C05348=1013.518,283.587,-142.989,169.129,53.074,160.196
C05349=1013.525,283.835,-143.018,169.134,53.067,160.195
C05350=1013.530,284.083,-143.047,169.141,53.060,160.195
C05351=1013.535,284.331,-143.077,169.146,53.053,160.195
C05352=1013.541,284.579,-143.107,169.151,53.046,160.194
C05353=1013.546,284.827,-143.137,169.157,53.039,160.194
C05354=1013.552,285.076,-143.167,169.163,53.032,160.193
C05355=1013.558,285.324,-143.197,169.169,53.025,160.193
C05356=1013.563,285.572,-143.227,169.174,53.018,160.192
C05357=1013.569,285.820,-143.257,169.181,53.011,160.192
C05358=1013.575,286.068,-143.287,169.186,53.004,160.192
C05359=1013.580,286.317,-143.316,169.192,52.997,160.191
C05360=1013.585,286.564,-143.346,169.198,52.990,160.191
C05361=1013.591,286.812,-143.376,169.204,52.983,160.191
C05362=1013.597,287.060,-143.406,169.209,52.976,160.190
C05363=1013.602,287.309,-143.436,169.216,52.969,160.190
C05364=1013.608,287.557,-143.466,169.222,52.962,160.190
C05365=1013.613,287.805,-143.496,169.227,52.955,160.189
C05366=1013.619,288.053,-143.526,169.233,52.949,160.189
C05367=1013.625,288.301,-143.556,169.239,52.941,160.188
C05368=1013.631,288.549,-143.586,169.245,52.935,160.188
C05369=1013.636,288.797,-143.617,169.250,52.928,160.187
C05370=1013.642,289.045,-143.646,169.257,52.921,160.187
C05371=1013.648,289.293,-143.676,169.263,52.915,160.187
C05372=1013.653,289.542,-143.706,169.268,52.908,160.187
C05373=1013.659,289.789,-143.736,169.274,52.901,160.186
C05374=1013.665,290.037,-143.767,169.280,52.894,160.186
C05375=1013.671,290.286,-143.798,169.286,52.887,160.186
C05376=1013.677,290.534,-143.827,169.292,52.881,160.185
C05377=1013.683,290.782,-143.858,169.298,52.873,160.185
C05378=1013.688,291.030,-143.888,169.304,52.867,160.185
C05379=1013.694,291.278,-143.918,169.310,52.861,160.184
C05380=1013.699,291.526,-143.949,169.316,52.854,160.184
C05381=1013.705,291.774,-143.979,169.322,52.847,160.184
C05382=1013.711,292.022,-144.009,169.328,52.840,160.183
C05383=1013.716,292.270,-144.040,169.334,52.834,160.183
C05384=1013.722,292.518,-144.070,169.339,52.827,160.183
C05385=1013.729,292.783,-144.103,169.346,52.820,160.182
C05386=1013.735,293.049,-144.136,169.353,52.813,160.182
C05387=1013.740,293.314,-144.169,169.359,52.806,160.182
C05388=1013.746,293.580,-144.202,169.365,52.799,160.181
C05389=1013.752,293.828,-144.233,169.372,52.792,160.181
C05390=1013.757,294.076,-144.264,169.377,52.786,160.181
C05391=1013.763,294.324,-144.295,169.383,52.780,160.181
C05392=1013.768,294.572,-144.326,169.389,52.773,160.180
C05393=1013.774,294.820,-144.356,169.395,52.767,160.180
C05394=1013.779,295.068,-144.387,169.402,52.760,160.180
C05395=1013.785,295.316,-144.418,169.407,52.754,160.179
C05396=1013.791,295.564,-144.450,169.413,52.747,160.179
C05397=1013.797,295.812,-144.480,169.419,52.741,160.179
C05398=1013.802,296.060,-144.511,169.425,52.734,160.179
C05399=1013.808,296.308,-144.542,169.431,52.728,160.178
C05400=1013.814,296.556,-144.573,169.438,52.721,160.178
C05401=1013.820,296.804,-144.604,169.444,52.716,160.178
C05402=1013.825,297.052,-144.635,169.450,52.709,160.178
C05403=1013.831,297.300,-144.666,169.455,52.703,160.177
C05404=1013.837,297.548,-144.698,169.461,52.696,160.177
C05405=1013.843,297.796,-144.728,169.468,52.690,160.177
C05406=1013.848,298.044,-144.759,169.474,52.683,160.177
C05407=1013.854,298.292,-144.790,169.480,52.678,160.177
C05408=1013.859,298.540,-144.821,169.486,52.671,160.176
C05409=1013.866,298.788,-144.853,169.492,52.665,160.176
C05410=1013.871,299.036,-144.884,169.499,52.658,160.176
C05411=1013.877,299.283,-144.915,169.505,52.652,160.176
C05412=1013.883,299.532,-144.946,169.511,52.646,160.175
C05413=1013.889,299.779,-144.977,169.517,52.640,160.175
C05414=1013.895,300.028,-145.008,169.523,52.634,160.175
C05415=1013.900,300.275,-145.040,169.529,52.627,160.175
C05416=1013.907,300.523,-145.072,169.535,52.621,160.175
C05417=1013.912,300.771,-145.102,169.542,52.615,160.174
C05418=1013.918,301.019,-145.134,169.548,52.609,160.174
C05419=1013.924,301.267,-145.165,169.553,52.602,160.174
C05420=1013.930,301.515,-145.196,169.560,52.597,160.174
C05421=1013.936,301.763,-145.228,169.566,52.590,160.174
C05422=1013.942,302.011,-145.258,169.573,52.584,160.174
C05423=1013.948,302.259,-145.290,169.579,52.578,160.173
C05424=1013.955,302.507,-145.322,169.585,52.572,160.173
C05425=1013.960,302.754,-145.353,169.591,52.566,160.173
C05426=1013.966,303.003,-145.384,169.597,52.559,160.173
C05427=1013.972,303.250,-145.416,169.604,52.553,160.173
C05428=1013.978,303.498,-145.447,169.610,52.547,160.172
C05429=1013.984,303.746,-145.479,169.616,52.541,160.172
C05430=1013.990,303.994,-145.510,169.622,52.535,160.172
C05431=1013.996,304.243,-145.542,169.629,52.529,160.172
C05432=1014.002,304.490,-145.573,169.635,52.523,160.172
C05433=1014.008,304.738,-145.605,169.641,52.517,160.171
C05434=1014.014,304.985,-145.636,169.647,52.511,160.171
C05435=1014.020,305.233,-145.668,169.653,52.505,160.171
C05436=1014.026,305.482,-145.700,169.660,52.498,160.171
C05437=1014.033,305.729,-145.731,169.667,52.493,160.171
C05438=1014.039,305.977,-145.763,169.672,52.486,160.171
C05439=1014.045,306.225,-145.794,169.679,52.481,160.171
C05440=1014.051,306.473,-145.826,169.686,52.475,160.171
C05441=1014.057,306.720,-145.857,169.692,52.468,160.170
C05442=1014.063,306.969,-145.889,169.698,52.463,160.170
C05443=1014.070,307.216,-145.921,169.704,52.457,160.170
C05444=1014.075,307.464,-145.953,169.711,52.451,160.170
C05445=1014.083,307.748,-145.989,169.719,52.444,160.170
C05446=1014.090,308.032,-146.025,169.725,52.437,160.170
C05447=1014.097,308.316,-146.062,169.733,52.430,160.170
C05448=1014.104,308.600,-146.098,169.740,52.424,160.169
C05449=1014.111,308.846,-146.130,169.746,52.418,160.169
C05450=1014.117,309.094,-146.161,169.753,52.412,160.169
C05451=1014.123,309.343,-146.193,169.760,52.406,160.169
C05452=1014.128,309.590,-146.226,169.766,52.401,160.169
C05453=1014.134,309.838,-146.258,169.772,52.395,160.169
C05454=1014.141,310.086,-146.291,169.779,52.389,160.169
C05455=1014.147,310.333,-146.324,169.785,52.384,160.169
C05456=1014.153,310.581,-146.356,169.792,52.379,160.169
C05457=1014.158,310.829,-146.389,169.798,52.373,160.169
C05458=1014.164,311.077,-146.421,169.804,52.367,160.169
C05459=1014.170,311.324,-146.453,169.811,52.362,160.169
C05460=1014.176,311.572,-146.486,169.817,52.356,160.169
C05461=1014.182,311.820,-146.518,169.824,52.350,160.169
C05462=1014.189,312.068,-146.551,169.831,52.345,160.169
C05463=1014.194,312.315,-146.584,169.837,52.339,160.169
C05464=1014.200,312.563,-146.616,169.843,52.333,160.169
C05465=1014.206,312.811,-146.649,169.850,52.328,160.169
C05466=1014.212,313.058,-146.681,169.856,52.323,160.169
C05467=1014.218,313.306,-146.714,169.863,52.317,160.169
C05468=1014.224,313.554,-146.746,169.869,52.311,160.169
C05469=1014.230,313.802,-146.780,169.876,52.306,160.169
C05470=1014.236,314.050,-146.812,169.883,52.300,160.169
C05471=1014.243,314.297,-146.845,169.889,52.295,160.169
C05472=1014.249,314.545,-146.878,169.896,52.290,160.169
C05473=1014.255,314.792,-146.911,169.902,52.284,160.169
C05474=1014.261,315.040,-146.944,169.909,52.278,160.169
C05475=1014.267,315.289,-146.976,169.915,52.273,160.169
C05476=1014.273,315.536,-147.009,169.922,52.268,160.169
C05477=1014.279,315.784,-147.041,169.928,52.263,160.169
C05478=1014.286,316.031,-147.074,169.936,52.257,160.169
C05479=1014.292,316.279,-147.107,169.942,52.252,160.169
C05480=1014.297,316.527,-147.140,169.949,52.246,160.169
C05481=1014.304,316.775,-147.173,169.955,52.241,160.169
C05482=1014.311,317.023,-147.206,169.962,52.236,160.169
C05483=1014.317,317.270,-147.239,169.968,52.231,160.169
C05484=1014.323,317.518,-147.272,169.975,52.225,160.169
C05485=1014.329,317.766,-147.305,169.982,52.220,160.169
C05486=1014.335,318.013,-147.338,169.989,52.214,160.169
C05487=1014.342,318.260,-147.371,169.995,52.209,160.169
C05488=1014.348,318.509,-147.404,170.002,52.203,160.169
C05489=1014.355,318.756,-147.437,170.008,52.198,160.169
C05490=1014.360,319.004,-147.470,170.015,52.193,160.169
C05491=1014.367,319.252,-147.503,170.022,52.187,160.169
C05492=1014.374,319.499,-147.537,170.029,52.182,160.169
C05493=1014.380,319.747,-147.570,170.036,52.177,160.170
C05494=1014.386,319.995,-147.602,170.042,52.172,160.169
C05495=1014.392,320.243,-147.636,170.049,52.167,160.170
C05496=1014.399,320.490,-147.669,170.056,52.162,160.170
C05497=1014.405,320.738,-147.702,170.063,52.156,160.170
C05498=1014.412,320.985,-147.735,170.070,52.151,160.170
C05499=1014.419,321.233,-147.769,170.076,52.146,160.170
C05500=1014.425,321.481,-147.802,170.083,52.141,160.170
C05501=1014.431,321.729,-147.835,170.090,52.136,160.170
C05502=1014.438,321.976,-147.869,170.096,52.131,160.170
C05503=1014.444,322.224,-147.901,170.104,52.125,160.170
C05504=1014.452,322.472,-147.935,170.110,52.120,160.170
C05505=1014.458,322.761,-147.974,170.118,52.114,160.171
C05506=1014.466,323.050,-148.013,170.126,52.108,160.171
C05507=1014.474,323.339,-148.052,170.135,52.102,160.171
C05508=1014.481,323.628,-148.091,170.143,52.096,160.171
C05509=1014.488,323.876,-148.124,170.149,52.091,160.171
C05510=1014.495,324.123,-148.158,170.156,52.086,160.171
C05511=1014.501,324.372,-148.191,170.164,52.081,160.171
C05512=1014.507,324.619,-148.225,170.170,52.076,160.172
C05513=1014.515,324.867,-148.259,170.177,52.071,160.172
C05514=1014.521,325.114,-148.291,170.184,52.066,160.172
C05515=1014.528,325.362,-148.325,170.192,52.061,160.172
C05516=1014.535,325.609,-148.359,170.198,52.056,160.172
C05517=1014.541,325.857,-148.392,170.205,52.051,160.172
C05518=1014.547,326.104,-148.426,170.212,52.046,160.172
C05519=1014.554,326.352,-148.460,170.219,52.042,160.173
C05520=1014.560,326.600,-148.495,170.226,52.037,160.173
C05521=1014.567,326.847,-148.528,170.233,52.031,160.173
C05522=1014.573,327.095,-148.563,170.240,52.026,160.173
C05523=1014.579,327.343,-148.597,170.247,52.022,160.174
C05524=1014.586,327.590,-148.631,170.254,52.017,160.174
C05525=1014.593,327.838,-148.665,170.261,52.012,160.174
C05526=1014.599,328.085,-148.699,170.268,52.008,160.174
C05527=1014.606,328.333,-148.733,170.275,52.003,160.174
C05528=1014.612,328.580,-148.768,170.283,51.998,160.175
C05529=1014.619,328.828,-148.802,170.290,51.993,160.175
C05530=1014.626,329.075,-148.836,170.296,51.988,160.175
C05531=1014.632,329.323,-148.870,170.303,51.984,160.175
C05532=1014.638,329.571,-148.904,170.310,51.979,160.175
C05533=1014.645,329.818,-148.938,170.318,51.974,160.176
C05534=1014.652,330.066,-148.973,170.325,51.969,160.176
C05535=1014.658,330.313,-149.007,170.332,51.965,160.176
C05536=1014.665,330.561,-149.041,170.339,51.960,160.176
C05537=1014.672,330.809,-149.076,170.346,51.956,160.177
C05538=1014.678,331.056,-149.111,170.353,51.951,160.177
C05539=1014.686,331.304,-149.145,170.361,51.946,160.177
C05540=1014.691,331.551,-149.179,170.368,51.942,160.178
C05541=1014.698,331.798,-149.214,170.375,51.937,160.178
C05542=1014.705,332.046,-149.248,170.382,51.933,160.178
C05543=1014.712,332.293,-149.283,170.389,51.928,160.178
C05544=1014.719,332.541,-149.317,170.397,51.923,160.178
C05545=1014.725,332.789,-149.352,170.404,51.919,160.179
C05546=1014.731,333.036,-149.386,170.411,51.914,160.179
C05547=1014.738,333.283,-149.421,170.418,51.910,160.179
C05548=1014.745,333.531,-149.457,170.425,51.905,160.180
C05549=1014.751,333.779,-149.491,170.433,51.901,160.180
C05550=1014.759,334.026,-149.526,170.440,51.896,160.180
C05551=1014.766,334.273,-149.561,170.448,51.892,160.181
C05552=1014.772,334.521,-149.595,170.455,51.888,160.181
C05553=1014.779,334.769,-149.630,170.462,51.883,160.181
C05554=1014.786,335.016,-149.665,170.470,51.878,160.182
C05555=1014.792,335.263,-149.700,170.477,51.874,160.182
C05556=1014.799,335.511,-149.735,170.484,51.870,160.182
C05557=1014.806,335.759,-149.770,170.491,51.865,160.182
C05558=1014.812,336.006,-149.805,170.498,51.861,160.183
C05559=1014.819,336.253,-149.840,170.506,51.856,160.183
C05560=1014.826,336.501,-149.875,170.513,51.852,160.184
C05561=1014.833,336.748,-149.911,170.521,51.848,160.184
C05562=1014.839,336.995,-149.946,170.528,51.843,160.184
C05563=1014.846,337.243,-149.980,170.535,51.839,160.185
C05564=1014.853,337.491,-150.015,170.543,51.834,160.185
C05565=1014.861,337.776,-150.056,170.551,51.830,160.185
C05566=1014.869,338.060,-150.097,170.560,51.825,160.186
C05567=1014.877,338.345,-150.136,170.569,51.820,160.186
C05568=1014.885,338.630,-150.177,170.578,51.815,160.187
C05569=1014.892,338.878,-150.212,170.585,51.811,160.187
C05570=1014.899,339.125,-150.248,170.592,51.807,160.187
C05571=1014.905,339.372,-150.284,170.600,51.803,160.188
C05572=1014.912,339.619,-150.319,170.608,51.798,160.188
C05573=1014.919,339.867,-150.355,170.615,51.794,160.189
C05574=1014.926,340.114,-150.390,170.623,51.790,160.189
C05575=1014.933,340.362,-150.426,170.630,51.786,160.190
C05576=1014.940,340.609,-150.461,170.638,51.781,160.190
C05577=1014.946,340.856,-150.497,170.645,51.778,160.191
C05578=1014.954,341.104,-150.533,170.653,51.773,160.191
C05579=1014.960,341.351,-150.568,170.660,51.770,160.191
C05580=1014.967,341.598,-150.604,170.668,51.765,160.192
C05581=1014.975,341.846,-150.639,170.675,51.761,160.192
C05582=1014.981,342.093,-150.676,170.683,51.757,160.193
C05583=1014.988,342.341,-150.711,170.690,51.753,160.193
C05584=1014.996,342.588,-150.747,170.699,51.749,160.194
C05585=1015.002,342.835,-150.782,170.706,51.745,160.194
C05586=1015.009,343.083,-150.819,170.714,51.741,160.194
C05587=1015.016,343.330,-150.855,170.721,51.737,160.195
C05588=1015.023,343.577,-150.890,170.729,51.733,160.195
C05589=1015.030,343.825,-150.927,170.737,51.729,160.196
C05590=1015.037,344.072,-150.963,170.744,51.726,160.197
C05591=1015.044,344.319,-150.998,170.753,51.721,160.197
C05592=1015.052,344.567,-151.034,170.760,51.717,160.197
C05593=1015.058,344.814,-151.070,170.768,51.714,160.198
C05594=1015.066,345.061,-151.107,170.776,51.709,160.198
C05595=1015.072,345.309,-151.142,170.783,51.705,160.199
C05596=1015.080,345.556,-151.178,170.791,51.702,160.199
C05597=1015.086,345.803,-151.214,170.799,51.698,160.200
C05598=1015.094,346.050,-151.251,170.807,51.694,160.201
C05599=1015.101,346.297,-151.286,170.814,51.690,160.201
C05600=1015.108,346.545,-151.323,170.822,51.686,160.201
C05601=1015.116,346.792,-151.359,170.830,51.682,160.202
C05602=1015.122,347.039,-151.396,170.838,51.679,160.203
C05603=1015.130,347.287,-151.432,170.846,51.675,160.203
C05604=1015.137,347.534,-151.468,170.854,51.671,160.204
C05605=1015.144,347.781,-151.505,170.862,51.667,160.204
C05606=1015.151,348.028,-151.541,170.869,51.664,160.205
C05607=1015.158,348.276,-151.577,170.878,51.660,160.206
C05608=1015.165,348.523,-151.615,170.886,51.656,160.206
C05609=1015.172,348.770,-151.651,170.893,51.652,160.207
C05610=1015.179,349.018,-151.688,170.902,51.649,160.207
C05611=1015.187,349.265,-151.724,170.909,51.645,160.208
C05612=1015.193,349.511,-151.761,170.917,51.641,160.208
C05613=1015.201,349.759,-151.797,170.926,51.638,160.209
C05614=1015.208,350.007,-151.834,170.933,51.634,160.210
C05615=1015.216,350.253,-151.871,170.942,51.630,160.210
C05616=1015.222,350.500,-151.907,170.950,51.627,160.211
C05617=1015.230,350.747,-151.944,170.957,51.623,160.211
C05618=1015.237,350.995,-151.981,170.966,51.620,160.212
C05619=1015.245,351.243,-152.017,170.974,51.616,160.213
C05620=1015.252,351.490,-152.055,170.981,51.612,160.213
C05621=1015.259,351.736,-152.091,170.990,51.609,160.214
C05622=1015.266,351.984,-152.128,170.998,51.605,160.215
C05623=1015.274,352.231,-152.166,171.006,51.601,160.215
C05624=1015.281,352.478,-152.202,171.014,51.598,160.216
C05625=1015.290,352.760,-152.244,171.024,51.594,160.217
C05626=1015.299,353.042,-152.287,171.033,51.590,160.217
C05627=1015.307,353.325,-152.329,171.043,51.586,160.218
C05628=1015.315,353.607,-152.371,171.052,51.582,160.219
C05629=1015.322,353.854,-152.408,171.060,51.579,160.220
C05630=1015.330,354.100,-152.445,171.068,51.575,160.220
C05631=1015.337,354.348,-152.483,171.077,51.572,160.221
C05632=1015.344,354.595,-152.520,171.084,51.568,160.222
C05633=1015.352,354.842,-152.558,171.093,51.565,160.222
C05634=1015.360,355.089,-152.595,171.101,51.561,160.223
C05635=1015.367,355.336,-152.632,171.110,51.558,160.224
C05636=1015.374,355.584,-152.669,171.118,51.555,160.224
C05637=1015.382,355.831,-152.707,171.126,51.551,160.225
C05638=1015.390,356.078,-152.745,171.134,51.548,160.226
C05639=1015.397,356.325,-152.782,171.143,51.545,160.227
C05640=1015.405,356.572,-152.820,171.151,51.542,160.227
C05641=1015.412,356.819,-152.857,171.160,51.538,160.228
C05642=1015.420,357.066,-152.894,171.168,51.535,160.229
C05643=1015.427,357.313,-152.932,171.177,51.532,160.230
C05644=1015.434,357.560,-152.969,171.185,51.529,160.230
C05645=1015.442,357.807,-153.008,171.194,51.525,160.231
C05646=1015.450,358.054,-153.045,171.202,51.522,160.232
C05647=1015.458,358.301,-153.082,171.211,51.519,160.233
C05648=1015.465,358.548,-153.120,171.219,51.516,160.233
C05649=1015.472,358.795,-153.158,171.227,51.512,160.234
C05650=1015.480,359.043,-153.196,171.236,51.510,160.235
C05651=1015.488,359.289,-153.234,171.245,51.506,160.236
C05652=1015.495,359.536,-153.272,171.253,51.503,160.237
C05653=1015.503,359.783,-153.310,171.262,51.500,160.237
C05654=1015.510,360.030,-153.348,171.270,51.497,160.238
C05655=1015.518,360.277,-153.386,171.279,51.494,160.239
C05656=1015.525,360.524,-153.424,171.287,51.491,160.240
C05657=1015.533,360.771,-153.462,171.296,51.487,160.241
C05658=1015.541,361.018,-153.501,171.304,51.485,160.242
C05659=1015.548,361.265,-153.539,171.313,51.482,160.242
C05660=1015.556,361.512,-153.576,171.322,51.478,160.243
C05661=1015.563,361.759,-153.616,171.330,51.475,160.244
C05662=1015.571,362.006,-153.654,171.339,51.472,160.245
C05663=1015.579,362.253,-153.692,171.347,51.469,160.246
C05664=1015.586,362.500,-153.730,171.356,51.466,160.247
C05665=1015.594,362.747,-153.768,171.366,51.463,160.248
C05666=1015.602,362.994,-153.807,171.374,51.460,160.248
C05667=1015.609,363.240,-153.845,171.383,51.457,160.249
C05668=1015.617,363.488,-153.884,171.391,51.455,160.250
C05669=1015.625,363.734,-153.922,171.400,51.451,160.251
C05670=1015.633,363.981,-153.960,171.410,51.449,160.252
C05671=1015.641,364.228,-153.999,171.418,51.446,160.253
C05672=1015.649,364.475,-154.037,171.427,51.443,160.254
C05673=1015.657,364.722,-154.076,171.436,51.440,160.255
C05674=1015.665,364.969,-154.114,171.444,51.437,160.256
C05675=1015.673,365.216,-154.153,171.453,51.434,160.256
C05676=1015.680,365.463,-154.191,171.463,51.431,160.257
C05677=1015.689,365.709,-154.230,171.471,51.429,160.258
C05678=1015.696,365.957,-154.270,171.480,51.425,160.259
C05679=1015.704,366.203,-154.308,171.489,51.423,160.260
C05680=1015.712,366.450,-154.346,171.499,51.420,160.261
C05681=1015.720,366.697,-154.386,171.507,51.417,160.262
C05682=1015.728,366.944,-154.424,171.516,51.414,160.263
C05683=1015.736,367.191,-154.463,171.526,51.412,160.264
C05684=1015.744,367.437,-154.502,171.534,51.409,160.265
C05685=1015.753,367.727,-154.548,171.545,51.406,160.266
C05686=1015.763,368.017,-154.594,171.556,51.403,160.267
C05687=1015.772,368.307,-154.639,171.566,51.400,160.268
C05688=1015.781,368.596,-154.685,171.577,51.396,160.270
C05689=1015.789,368.843,-154.725,171.586,51.394,160.271
C05690=1015.797,369.090,-154.764,171.595,51.391,160.272
C05691=1015.806,369.336,-154.804,171.605,51.388,160.273
C05692=1015.813,369.584,-154.843,171.613,51.386,160.274
C05693=1015.821,369.831,-154.882,171.623,51.383,160.275
C05694=1015.829,370.077,-154.922,171.632,51.380,160.276
C05695=1015.837,370.323,-154.961,171.642,51.378,160.277
C05696=1015.845,370.570,-155.000,171.651,51.376,160.278
C05697=1015.853,370.817,-155.040,171.660,51.373,160.279
C05698=1015.861,371.064,-155.079,171.669,51.371,160.280
C05699=1015.869,371.311,-155.119,171.678,51.368,160.281
C05700=1015.878,371.558,-155.158,171.688,51.366,160.282
C05701=1015.886,371.804,-155.197,171.698,51.363,160.283
C05702=1015.894,372.051,-155.237,171.707,51.360,160.284
C05703=1015.902,372.298,-155.277,171.715,51.358,160.285
C05704=1015.911,372.544,-155.317,171.725,51.356,160.287
C05705=1015.919,372.791,-155.357,171.735,51.353,160.288
C05706=1015.927,373.037,-155.396,171.744,51.351,160.289
C05707=1015.935,373.284,-155.436,171.754,51.348,160.290
C05708=1015.943,373.531,-155.475,171.763,51.346,160.291
C05709=1015.952,373.778,-155.515,171.773,51.343,160.292
C05710=1015.960,374.024,-155.556,171.782,51.341,160.293
C05711=1015.969,374.271,-155.595,171.792,51.339,160.294
C05712=1015.977,374.518,-155.635,171.801,51.336,160.295
C05713=1015.985,374.764,-155.675,171.811,51.334,160.297
C05714=1015.994,375.011,-155.715,171.821,51.332,160.298
C05715=1016.002,375.258,-155.754,171.830,51.329,160.299
C05716=1016.011,375.504,-155.795,171.840,51.327,160.300
C05717=1016.019,375.751,-155.834,171.850,51.325,160.302
C05718=1016.027,375.998,-155.875,171.859,51.322,160.303
C05719=1016.036,376.244,-155.915,171.868,51.320,160.304
C05720=1016.044,376.491,-155.955,171.878,51.318,160.305
C05721=1016.052,376.737,-155.996,171.888,51.316,160.306
C05722=1016.060,376.984,-156.037,171.898,51.314,160.307
C05723=1016.069,377.230,-156.077,171.907,51.311,160.308
C05724=1016.077,377.476,-156.118,171.917,51.309,160.310
C05725=1016.085,377.724,-156.158,171.927,51.307,160.311
C05726=1016.093,377.970,-156.199,171.937,51.304,160.312
C05727=1016.102,378.216,-156.239,171.947,51.302,160.314
C05728=1016.111,378.463,-156.280,171.957,51.300,160.315
C05729=1016.119,378.709,-156.320,171.967,51.298,160.316
C05730=1016.128,378.956,-156.361,171.977,51.296,160.317
C05731=1016.136,379.202,-156.401,171.986,51.294,160.319
C05732=1016.145,379.449,-156.442,171.997,51.292,160.320
C05733=1016.153,379.696,-156.483,172.006,51.290,160.321
C05734=1016.163,379.942,-156.524,172.016,51.288,160.323
C05735=1016.171,380.188,-156.565,172.026,51.286,160.324
C05736=1016.179,380.435,-156.606,172.036,51.284,160.325
C05737=1016.187,380.681,-156.646,172.047,51.282,160.327
C05738=1016.197,380.928,-156.687,172.057,51.280,160.328
C05739=1016.206,381.174,-156.728,172.067,51.278,160.329
C05740=1016.214,381.421,-156.769,172.076,51.276,160.330
C05741=1016.222,381.668,-156.810,172.087,51.274,160.332
C05742=1016.231,381.913,-156.851,172.097,51.272,160.333
C05743=1016.240,382.160,-156.892,172.108,51.270,160.335
C05744=1016.249,382.407,-156.933,172.117,51.268,160.336
C05745=1016.260,382.719,-156.985,172.130,51.265,160.338
C05746=1016.271,383.031,-157.037,172.143,51.263,160.339
C05747=1016.282,383.343,-157.090,172.156,51.261,160.341
C05748=1016.294,383.656,-157.141,172.169,51.258,160.343
C05749=1016.303,383.903,-157.183,172.179,51.256,160.344
C05750=1016.311,384.148,-157.224,172.190,51.254,160.346
C05751=1016.321,384.395,-157.265,172.201,51.253,160.347
C05752=1016.330,384.641,-157.307,172.210,51.251,160.348
C05753=1016.338,384.888,-157.348,172.222,51.249,160.350
C05754=1016.347,385.134,-157.390,172.232,51.247,160.351
C05755=1016.356,385.381,-157.432,172.242,51.246,160.353
C05756=1016.365,385.627,-157.473,172.253,51.243,160.354
C05757=1016.374,385.873,-157.515,172.263,51.242,160.356
C05758=1016.383,386.120,-157.557,172.273,51.240,160.357
C05759=1016.392,386.366,-157.599,172.284,51.238,160.359
C05760=1016.401,386.612,-157.640,172.295,51.237,160.360
C05761=1016.409,386.858,-157.682,172.305,51.235,160.362
C05762=1016.419,387.105,-157.724,172.316,51.234,160.363
C05763=1016.428,387.351,-157.765,172.326,51.232,160.365
C05764=1016.437,387.598,-157.807,172.337,51.230,160.366
C05765=1016.446,387.844,-157.850,172.348,51.229,160.368
C05766=1016.455,388.090,-157.891,172.359,51.227,160.369
C05767=1016.464,388.336,-157.934,172.369,51.226,160.371
C05768=1016.473,388.582,-157.975,172.380,51.224,160.372
C05769=1016.482,388.828,-158.017,172.391,51.222,160.374
C05770=1016.490,389.074,-158.060,172.401,51.221,160.375
C05771=1016.499,389.321,-158.102,172.413,51.220,160.377
C05772=1016.509,389.567,-158.145,172.423,51.218,160.378
C05773=1016.519,389.813,-158.187,172.434,51.216,160.380
C05774=1016.527,390.059,-158.229,172.446,51.215,160.382
C05775=1016.537,390.305,-158.271,172.456,51.213,160.383
C05776=1016.547,390.552,-158.314,172.467,51.212,160.385
C05777=1016.555,390.798,-158.356,172.478,51.210,160.386
C05778=1016.564,391.044,-158.399,172.489,51.209,160.388
C05779=1016.574,391.290,-158.442,172.499,51.208,160.390
C05780=1016.583,391.536,-158.484,172.511,51.206,160.391
C05781=1016.592,391.783,-158.526,172.522,51.204,160.393
C05782=1016.602,392.029,-158.569,172.533,51.203,160.395
C05783=1016.610,392.275,-158.612,172.544,51.202,160.396
C05784=1016.620,392.522,-158.654,172.555,51.200,160.398
C05785=1016.630,392.767,-158.698,172.566,51.199,160.400
C05786=1016.639,393.012,-158.740,172.578,51.198,160.401
C05787=1016.648,393.259,-158.783,172.589,51.197,160.403
C05788=1016.657,393.505,-158.826,172.599,51.195,160.405
C05789=1016.667,393.751,-158.869,172.611,51.194,160.406
C05790=1016.676,393.997,-158.912,172.623,51.192,160.408
C05791=1016.686,394.243,-158.955,172.633,51.192,160.410
C05792=1016.696,394.490,-158.998,172.645,51.190,160.412
C05793=1016.704,394.736,-159.041,172.656,51.189,160.413
C05794=1016.714,394.982,-159.084,172.668,51.188,160.415
C05795=1016.724,395.227,-159.127,172.680,51.186,160.417
C05796=1016.733,395.473,-159.171,172.690,51.185,160.419
C05797=1016.743,395.720,-159.214,172.702,51.184,160.420
C05798=1016.752,395.965,-159.257,172.713,51.183,160.422
C05799=1016.761,396.212,-159.300,172.725,51.182,160.424
C05800=1016.772,396.458,-159.344,172.737,51.181,160.426
C05801=1016.782,396.703,-159.387,172.749,51.179,160.428
C05802=1016.790,396.949,-159.430,172.760,51.178,160.429
C05803=1016.800,397.195,-159.474,172.771,51.178,160.431
C05804=1016.810,397.441,-159.518,172.783,51.176,160.433
C05805=1016.824,397.787,-159.579,172.799,51.175,160.436
C05806=1016.837,398.133,-159.641,172.816,51.174,160.438
C05807=1016.851,398.479,-159.702,172.832,51.172,160.441
C05808=1016.865,398.826,-159.764,172.849,51.170,160.443
C05809=1016.874,399.071,-159.807,172.861,51.170,160.445
C05810=1016.884,399.318,-159.851,172.873,51.169,160.447
C05811=1016.894,399.563,-159.895,172.884,51.168,160.449
C05812=1016.904,399.809,-159.940,172.896,51.167,160.451
C05813=1016.914,400.055,-159.983,172.909,51.166,160.453
C05814=1016.923,400.301,-160.027,172.921,51.164,160.455
C05815=1016.934,400.547,-160.073,172.933,51.164,160.457
C05816=1016.943,400.793,-160.117,172.945,51.163,160.459
C05817=1016.953,401.038,-160.161,172.957,51.162,160.461
C05818=1016.963,401.285,-160.205,172.969,51.161,160.463
C05819=1016.973,401.530,-160.250,172.981,51.161,160.465
C05820=1016.983,401.776,-160.293,172.993,51.160,160.467
C05821=1016.992,402.021,-160.338,173.005,51.159,160.469
C05822=1017.002,402.268,-160.382,173.018,51.158,160.471
C05823=1017.012,402.514,-160.427,173.030,51.157,160.473
C05824=1017.023,402.759,-160.472,173.042,51.156,160.475
C05825=1017.032,403.004,-160.517,173.054,51.156,160.477
C05826=1017.042,403.251,-160.561,173.066,51.156,160.479
C05827=1017.053,403.497,-160.605,173.079,51.154,160.481
C05828=1017.062,403.742,-160.650,173.091,51.154,160.483
C05829=1017.072,403.988,-160.695,173.103,51.153,160.485
C05830=1017.083,404.233,-160.739,173.117,51.152,160.487
C05831=1017.093,404.479,-160.784,173.129,51.152,160.489
C05832=1017.103,404.724,-160.829,173.141,51.151,160.491
C05833=1017.113,404.971,-160.874,173.154,51.150,160.493
C05834=1017.123,405.216,-160.919,173.166,51.149,160.495
C05835=1017.134,405.461,-160.964,173.178,51.149,160.498
C05836=1017.144,405.707,-161.009,173.192,51.149,160.500
C05837=1017.155,405.953,-161.054,173.204,51.148,160.502
C05838=1017.165,406.198,-161.099,173.217,51.147,160.504
C05839=1017.175,406.444,-161.145,173.229,51.147,160.506
C05840=1017.186,406.690,-161.189,173.242,51.146,160.508
C05841=1016.824,404.675,-161.163,173.123,51.219,160.507
C05842=1016.814,404.429,-161.118,173.110,51.220,160.505
C05843=1016.804,404.183,-161.073,173.097,51.220,160.502
C05844=1016.793,403.938,-161.029,173.085,51.221,160.500
C05845=1016.784,403.692,-160.984,173.072,51.222,160.498
C05846=1016.773,403.446,-160.939,173.060,51.223,160.496
C05847=1016.763,403.201,-160.894,173.048,51.223,160.494
C05848=1016.753,402.955,-160.850,173.035,51.224,160.492
C05849=1016.744,402.709,-160.805,173.023,51.225,160.490
C05850=1016.733,402.463,-160.761,173.011,51.226,160.488
C05851=1016.723,402.217,-160.717,172.998,51.227,160.486
C05852=1016.714,401.972,-160.672,172.986,51.228,160.484
C05853=1016.704,401.726,-160.627,172.974,51.229,160.482
C05854=1016.694,401.480,-160.584,172.962,51.229,160.480
C05855=1016.684,401.235,-160.539,172.950,51.230,160.478
C05856=1016.675,400.989,-160.495,172.937,51.231,160.476
C05857=1016.664,400.744,-160.450,172.925,51.232,160.474
C05858=1016.654,400.497,-160.406,172.914,51.234,160.473
C05859=1016.645,400.251,-160.362,172.902,51.234,160.471
C05860=1016.634,400.005,-160.318,172.890,51.235,160.469
C05861=1016.625,399.759,-160.273,172.878,51.236,160.467
C05862=1016.615,399.513,-160.229,172.866,51.237,160.465
C05863=1016.605,399.267,-160.186,172.853,51.238,160.463
C05864=1016.596,399.021,-160.142,172.842,51.240,160.461
C05865=1016.586,398.776,-160.099,172.830,51.240,160.459
C05866=1016.574,398.464,-160.042,172.816,51.242,160.457
C05867=1016.561,398.152,-159.987,172.800,51.243,160.454
C05868=1016.550,397.839,-159.932,172.785,51.245,160.452
C05869=1016.537,397.528,-159.876,172.770,51.246,160.450
C05870=1016.527,397.282,-159.832,172.758,51.248,160.448
C05871=1016.518,397.036,-159.789,172.747,51.249,160.446
C05872=1016.508,396.790,-159.746,172.736,51.249,160.444
C05873=1016.498,396.544,-159.702,172.724,51.251,160.442
C05874=1016.489,396.297,-159.659,172.712,51.252,160.441
C05875=1016.479,396.052,-159.616,172.701,51.253,160.439
C05876=1016.470,395.805,-159.572,172.689,51.255,160.437
C05877=1016.460,395.560,-159.529,172.678,51.256,160.435
C05878=1016.451,395.314,-159.487,172.666,51.257,160.434
C05879=1016.441,395.068,-159.442,172.654,51.259,160.432
C05880=1016.431,394.821,-159.400,172.643,51.260,160.430
C05881=1016.422,394.576,-159.356,172.631,51.261,160.428
C05882=1016.412,394.330,-159.314,172.621,51.262,160.427
C05883=1016.403,394.084,-159.271,172.609,51.264,160.425
C05884=1016.394,393.837,-159.228,172.598,51.266,160.423
C05885=1016.384,393.592,-159.185,172.586,51.267,160.422
C05886=1016.375,393.345,-159.141,172.575,51.268,160.420
C05887=1016.366,393.100,-159.099,172.564,51.269,160.418
C05888=1016.356,392.853,-159.056,172.553,51.271,160.417
C05889=1016.347,392.607,-159.013,172.541,51.272,160.415
C05890=1016.338,392.361,-158.970,172.530,51.274,160.413
C05891=1016.328,392.115,-158.928,172.519,51.275,160.411
C05892=1016.320,391.869,-158.885,172.508,51.277,160.410
C05893=1016.310,391.622,-158.842,172.497,51.279,160.408
C05894=1016.301,391.377,-158.800,172.486,51.279,160.406
C05895=1016.292,391.130,-158.758,172.475,51.281,160.405
C05896=1016.282,390.884,-158.715,172.463,51.283,160.403
C05897=1016.273,390.638,-158.673,172.453,51.284,160.402
C05898=1016.263,390.392,-158.630,172.442,51.286,160.400
C05899=1016.254,390.145,-158.588,172.430,51.287,160.398
C05900=1016.245,389.899,-158.545,172.420,51.289,160.397
C05901=1016.237,389.653,-158.503,172.409,51.291,160.395
C05902=1016.227,389.407,-158.461,172.398,51.293,160.394
C05903=1016.218,389.161,-158.419,172.387,51.294,160.392
C05904=1016.209,388.914,-158.376,172.376,51.296,160.391
C05905=1016.200,388.668,-158.335,172.366,51.297,160.389
C05906=1016.190,388.422,-158.292,172.355,51.299,160.388
C05907=1016.181,388.176,-158.251,172.344,51.301,160.386
C05908=1016.173,387.930,-158.208,172.333,51.303,160.385
C05909=1016.164,387.683,-158.166,172.323,51.304,160.383
C05910=1016.155,387.437,-158.124,172.312,51.306,160.382
C05911=1016.146,387.191,-158.082,172.302,51.308,160.380
C05912=1016.137,386.944,-158.041,172.290,51.309,160.379
C05913=1016.128,386.698,-157.999,172.280,51.311,160.377
C05914=1016.119,386.452,-157.957,172.269,51.313,160.375
C05915=1016.110,386.206,-157.915,172.259,51.314,160.374
C05916=1016.101,385.959,-157.873,172.248,51.317,160.373
C05917=1016.092,385.713,-157.831,172.238,51.319,160.371
C05918=1016.083,385.467,-157.790,172.227,51.320,160.370
C05919=1016.075,385.220,-157.749,172.216,51.322,160.368
C05920=1016.065,384.974,-157.708,172.207,51.324,160.367
C05921=1016.057,384.728,-157.666,172.195,51.326,160.365
C05922=1016.048,384.482,-157.624,172.185,51.328,160.364
C05923=1016.039,384.235,-157.583,172.174,51.330,160.363
C05924=1016.030,383.988,-157.542,172.164,51.332,160.361
C05925=1016.020,383.742,-157.501,172.154,51.334,160.360
C05926=1016.010,383.427,-157.448,172.141,51.336,160.358
C05927=1015.998,383.113,-157.395,172.128,51.338,160.356
C05928=1015.987,382.798,-157.343,172.114,51.341,160.354
C05929=1015.975,382.483,-157.291,172.101,51.344,160.353
C05930=1015.967,382.236,-157.250,172.091,51.346,160.351
C05931=1015.958,381.991,-157.208,172.081,51.348,160.350
C05932=1015.950,381.744,-157.167,172.070,51.350,160.349
C05933=1015.940,381.497,-157.127,172.061,51.352,160.347
C05934=1015.932,381.251,-157.086,172.051,51.354,160.346
C05935=1015.923,381.004,-157.045,172.040,51.357,160.345
C05936=1015.915,380.758,-157.005,172.030,51.359,160.344
C05937=1015.906,380.511,-156.964,172.020,51.360,160.342
C05938=1015.898,380.266,-156.922,172.010,51.362,160.341
C05939=1015.889,380.019,-156.881,171.999,51.365,160.340
C05940=1015.880,379.772,-156.841,171.990,51.367,160.338
C05941=1015.872,379.526,-156.800,171.980,51.369,160.337
C05942=1015.864,379.279,-156.760,171.970,51.371,160.336
C05943=1015.855,379.032,-156.719,171.960,51.373,160.335
C05944=1015.846,378.787,-156.679,171.950,51.376,160.333
C05945=1015.838,378.540,-156.638,171.940,51.378,160.332
C05946=1015.830,378.293,-156.597,171.930,51.380,160.331
C05947=1015.820,378.047,-156.557,171.920,51.382,160.329
C05948=1015.812,377.800,-156.516,171.910,51.384,160.328
C05949=1015.805,377.553,-156.476,171.901,51.387,160.327
C05950=1015.796,377.306,-156.435,171.891,51.389,160.326
C05951=1015.787,377.060,-156.395,171.881,51.391,160.325
C05952=1015.779,376.814,-156.354,171.871,51.394,160.323
C05953=1015.771,376.567,-156.314,171.862,51.396,160.322
C05954=1015.763,376.320,-156.273,171.852,51.398,160.321
C05955=1015.754,376.074,-156.233,171.841,51.401,160.320
C05956=1015.746,375.827,-156.193,171.832,51.403,160.318
C05957=1015.738,375.581,-156.153,171.822,51.406,160.317
C05958=1015.729,375.334,-156.112,171.813,51.408,160.316
C05959=1015.721,375.088,-156.072,171.803,51.411,160.315
C05960=1015.713,374.841,-156.033,171.793,51.413,160.314
C05961=1015.705,374.595,-155.993,171.784,51.416,160.313
C05962=1015.696,374.348,-155.953,171.774,51.418,160.312
C05963=1015.687,374.101,-155.914,171.765,51.420,160.311
C05964=1015.679,373.854,-155.874,171.755,51.423,160.309
C05965=1015.671,373.608,-155.834,171.746,51.425,160.308
C05966=1015.662,373.361,-155.794,171.736,51.428,160.307
C05967=1015.655,373.114,-155.754,171.726,51.430,160.306
C05968=1015.646,372.868,-155.715,171.717,51.433,160.305
C05969=1015.638,372.621,-155.675,171.708,51.436,160.304
C05970=1015.630,372.374,-155.636,171.698,51.438,160.303
C05971=1015.621,372.128,-155.596,171.688,51.440,160.302
C05972=1015.614,371.881,-155.556,171.679,51.443,160.301
C05973=1015.605,371.634,-155.517,171.670,51.446,160.299
C05974=1015.598,371.387,-155.477,171.661,51.448,160.299
C05975=1015.589,371.141,-155.438,171.652,51.451,160.298
C05976=1015.581,370.894,-155.399,171.642,51.454,160.296
C05977=1015.573,370.647,-155.359,171.633,51.456,160.295
C05978=1015.564,370.401,-155.319,171.623,51.459,160.294
C05979=1015.557,370.154,-155.279,171.614,51.461,160.293
C05980=1015.549,369.906,-155.241,171.604,51.464,160.292
C05981=1015.541,369.661,-155.202,171.595,51.467,160.291
C05982=1015.533,369.414,-155.162,171.587,51.469,160.290
C05983=1015.525,369.166,-155.123,171.577,51.472,160.289
C05984=1015.516,368.920,-155.084,171.568,51.475,160.288
C05985=1015.509,368.673,-155.044,171.559,51.478,160.287
C05986=1015.500,368.381,-154.998,171.549,51.481,160.286
C05987=1015.491,368.089,-154.952,171.537,51.485,160.285
C05988=1015.481,367.797,-154.906,171.527,51.488,160.284
C05989=1015.471,367.505,-154.859,171.515,51.491,160.282
C05990=1015.464,367.258,-154.820,171.507,51.494,160.281
C05991=1015.456,367.011,-154.781,171.498,51.496,160.280
C05992=1015.448,366.765,-154.743,171.489,51.500,160.280
C05993=1015.440,366.518,-154.704,171.479,51.502,160.279
C05994=1015.431,366.271,-154.665,171.470,51.505,160.278
C05995=1015.424,366.024,-154.626,171.462,51.508,160.277
C05996=1015.416,365.777,-154.588,171.452,51.511,160.276
C05997=1015.408,365.530,-154.549,171.443,51.514,160.275
C05998=1015.400,365.284,-154.511,171.434,51.517,160.274
C05999=1015.392,365.036,-154.472,171.425,51.520,160.273
C06000=1015.384,364.790,-154.434,171.417,51.523,160.272
C06001=1015.376,364.543,-154.396,171.408,51.526,160.271
C06002=1015.369,364.296,-154.357,171.398,51.529,160.270
C06003=1015.361,364.049,-154.318,171.390,51.532,160.269
C06004=1015.353,363.801,-154.279,171.381,51.535,160.269
C06005=1015.346,363.555,-154.241,171.372,51.538,160.268
C06006=1015.338,363.308,-154.203,171.363,51.541,160.267
C06007=1015.330,363.061,-154.164,171.355,51.544,160.266
C06008=1015.322,362.815,-154.126,171.346,51.547,160.265
C06009=1015.314,362.567,-154.088,171.337,51.550,160.264
C06010=1015.307,362.321,-154.049,171.329,51.553,160.263
C06011=1015.299,362.073,-154.011,171.320,51.557,160.263
C06012=1015.291,361.826,-153.973,171.310,51.560,160.262
C06013=1015.284,361.580,-153.935,171.302,51.563,160.261
C06014=1015.275,361.333,-153.896,171.293,51.566,160.260
C06015=1015.268,361.086,-153.859,171.284,51.569,160.259
C06016=1015.261,360.839,-153.821,171.276,51.572,160.258
C06017=1015.253,360.591,-153.783,171.267,51.576,160.258
C06018=1015.245,360.345,-153.744,171.258,51.579,160.257
C06019=1015.238,360.098,-153.706,171.250,51.581,160.256
C06020=1015.230,359.851,-153.669,171.241,51.585,160.255
C06021=1015.223,359.604,-153.629,171.233,51.588,160.254
C06022=1015.216,359.356,-153.592,171.224,51.591,160.253
C06023=1015.208,359.110,-153.554,171.215,51.594,160.252
C06024=1015.201,358.863,-153.516,171.207,51.598,160.252
C06025=1015.194,358.616,-153.479,171.198,51.601,160.251
C06026=1015.185,358.369,-153.441,171.190,51.604,160.250
C06027=1015.178,358.122,-153.403,171.181,51.608,160.250
C06028=1015.170,357.874,-153.366,171.172,51.611,160.249
C06029=1015.163,357.627,-153.328,171.164,51.614,160.248
C06030=1015.155,357.381,-153.290,171.156,51.618,160.247
C06031=1015.148,357.134,-153.253,171.148,51.621,160.247
C06032=1015.140,356.886,-153.215,171.139,51.625,160.246
C06033=1015.133,356.639,-153.177,171.131,51.627,160.245
C06034=1015.125,356.392,-153.140,171.122,51.632,160.244
C06035=1015.117,356.145,-153.103,171.113,51.635,160.244
C06036=1015.110,355.898,-153.065,171.106,51.639,160.243
C06037=1015.103,355.651,-153.028,171.097,51.642,160.242
C06038=1015.095,355.404,-152.991,171.089,51.645,160.241
C06039=1015.088,355.157,-152.953,171.080,51.649,160.241
C06040=1015.080,354.910,-152.916,171.072,51.652,160.240
C06041=1015.073,354.663,-152.878,171.064,51.656,160.239
C06042=1015.065,354.415,-152.842,171.056,51.659,160.239
C06043=1015.058,354.168,-152.805,171.047,51.663,160.238
C06044=1015.051,353.921,-152.767,171.039,51.666,160.237
C06045=1015.044,353.674,-152.730,171.031,51.670,160.237
C06046=1015.035,353.390,-152.687,171.021,51.674,160.236
C06047=1015.027,353.105,-152.644,171.012,51.678,160.235
C06048=1015.018,352.821,-152.602,171.002,51.682,160.234
C06049=1015.010,352.536,-152.560,170.993,51.686,160.234
C06050=1015.003,352.289,-152.522,170.985,51.690,160.233
C06051=1014.995,352.042,-152.486,170.976,51.693,160.232
C06052=1014.988,351.795,-152.449,170.969,51.697,160.232
C06053=1014.981,351.548,-152.413,170.960,51.701,160.231
C06054=1014.973,351.301,-152.375,170.953,51.705,160.231
C06055=1014.966,351.053,-152.339,170.944,51.708,160.230
C06056=1014.958,350.806,-152.302,170.936,51.712,160.229
C06057=1014.951,350.559,-152.265,170.927,51.716,160.229
C06058=1014.944,350.312,-152.228,170.920,51.719,160.228
C06059=1014.937,350.065,-152.192,170.911,51.723,160.228
C06060=1014.930,349.817,-152.155,170.904,51.727,160.227
C06061=1014.922,349.570,-152.119,170.895,51.731,160.226
C06062=1014.915,349.323,-152.082,170.888,51.735,160.226
C06063=1014.908,349.075,-152.045,170.880,51.738,160.225
C06064=1014.901,348.829,-152.009,170.871,51.742,160.225
C06065=1014.894,348.581,-151.972,170.864,51.746,160.224
C06066=1014.886,348.334,-151.935,170.855,51.750,160.223
C06067=1014.880,348.087,-151.899,170.848,51.754,160.223
C06068=1014.872,347.840,-151.863,170.840,51.757,160.222
C06069=1014.865,347.592,-151.826,170.832,51.761,160.222
C06070=1014.858,347.345,-151.790,170.824,51.765,160.221
C06071=1014.851,347.097,-151.753,170.815,51.769,160.221
C06072=1014.844,346.851,-151.717,170.808,51.772,160.220
C06073=1014.837,346.603,-151.681,170.801,51.777,160.220
C06074=1014.830,346.356,-151.645,170.792,51.781,160.219
C06075=1014.823,346.109,-151.609,170.785,51.784,160.219
C06076=1014.816,345.862,-151.573,170.776,51.788,160.218
C06077=1014.809,345.614,-151.536,170.769,51.793,160.218
C06078=1014.802,345.367,-151.501,170.761,51.796,160.217
C06079=1014.794,345.119,-151.465,170.753,51.800,160.216
C06080=1014.788,344.872,-151.428,170.746,51.805,160.216
C06081=1014.780,344.625,-151.392,170.737,51.809,160.216
C06082=1014.773,344.377,-151.357,170.729,51.812,160.215
C06083=1014.766,344.130,-151.321,170.722,51.817,160.215
C06084=1014.759,343.883,-151.284,170.714,51.821,160.214
C06085=1014.753,343.636,-151.249,170.707,51.825,160.214
C06086=1014.745,343.388,-151.213,170.699,51.829,160.213
C06087=1014.738,343.141,-151.178,170.691,51.833,160.213
C06088=1014.732,342.894,-151.141,170.683,51.837,160.212
C06089=1014.724,342.646,-151.105,170.676,51.841,160.212
C06090=1014.717,342.399,-151.070,170.668,51.845,160.211
C06091=1014.710,342.152,-151.034,170.660,51.849,160.211
C06092=1014.704,341.904,-150.998,170.652,51.853,160.210
C06093=1014.697,341.656,-150.963,170.645,51.858,160.210
C06094=1014.690,341.410,-150.927,170.638,51.862,160.210
C06095=1014.682,341.162,-150.891,170.629,51.866,160.209
C06096=1014.675,340.915,-150.856,170.622,51.870,160.209
C06097=1014.669,340.667,-150.820,170.615,51.875,160.208
C06098=1014.663,340.420,-150.785,170.607,51.878,160.208
C06099=1014.656,340.172,-150.750,170.599,51.883,160.207
C06100=1014.648,339.925,-150.713,170.592,51.887,160.207
C06101=1014.641,339.678,-150.678,170.585,51.892,160.207
C06102=1014.635,339.430,-150.643,170.576,51.896,160.206
C06103=1014.629,339.183,-150.607,170.569,51.900,160.206
C06104=1014.621,338.936,-150.571,170.562,51.904,160.205
C06105=1014.615,338.689,-150.536,170.554,51.909,160.205
C06106=1014.607,338.401,-150.496,170.545,51.914,160.205
C06107=1014.598,338.114,-150.454,170.536,51.919,160.204
C06108=1014.590,337.826,-150.414,170.528,51.924,160.204
C06109=1014.582,337.540,-150.373,170.519,51.929,160.203
C06110=1014.576,337.292,-150.338,170.511,51.934,160.203
C06111=1014.569,337.044,-150.303,170.504,51.938,160.203
C06112=1014.562,336.797,-150.268,170.497,51.942,160.202
C06113=1014.556,336.550,-150.233,170.490,51.947,160.202
C06114=1014.549,336.302,-150.198,170.482,51.951,160.202
C06115=1014.542,336.055,-150.163,170.474,51.956,160.201
C06116=1014.535,335.808,-150.128,170.467,51.960,160.201
C06117=1014.529,335.560,-150.093,170.459,51.965,160.200
C06118=1014.521,335.312,-150.059,170.452,51.969,160.200
C06119=1014.515,335.065,-150.024,170.445,51.974,160.200
C06120=1014.508,334.818,-149.988,170.437,51.978,160.200
C06121=1014.501,334.570,-149.954,170.430,51.983,160.199
C06122=1014.495,334.322,-149.919,170.423,51.987,160.199
C06123=1014.488,334.075,-149.884,170.416,51.992,160.199
C06124=1014.481,333.827,-149.849,170.408,51.997,160.198
C06125=1014.475,333.580,-149.815,170.401,52.001,160.198
C06126=1014.469,333.332,-149.780,170.394,52.005,160.198
C06127=1014.462,333.085,-149.745,170.387,52.010,160.198
C06128=1014.455,332.838,-149.710,170.379,52.015,160.197
C06129=1014.449,332.590,-149.675,170.372,52.019,160.197
C06130=1014.442,332.342,-149.640,170.365,52.024,160.197
C06131=1014.435,332.095,-149.607,170.358,52.029,160.196
C06132=1014.429,331.847,-149.572,170.350,52.034,160.196
C06133=1014.422,331.600,-149.537,170.343,52.038,160.196
C06134=1014.415,331.352,-149.503,170.336,52.043,160.195
C06135=1014.408,331.104,-149.469,170.329,52.047,160.195
C06136=1014.402,330.858,-149.434,170.321,52.052,160.195
C06137=1014.395,330.610,-149.400,170.314,52.057,160.195
C06138=1014.389,330.362,-149.366,170.307,52.062,160.195
C06139=1014.382,330.114,-149.332,170.299,52.067,160.194
C06140=1014.375,329.868,-149.297,170.293,52.072,160.194
C06141=1014.369,329.620,-149.263,170.285,52.076,160.194
C06142=1014.362,329.372,-149.229,170.279,52.081,160.194
C06143=1014.356,329.125,-149.195,170.271,52.086,160.194
C06144=1014.349,328.877,-149.161,170.264,52.091,160.193
C06145=1014.343,328.629,-149.126,170.257,52.096,160.193
C06146=1014.336,328.382,-149.093,170.250,52.101,160.193
C06147=1014.330,328.134,-149.058,170.242,52.105,160.193
C06148=1014.324,327.887,-149.024,170.236,52.110,160.192
C06149=1014.317,327.639,-148.991,170.229,52.115,160.192
C06150=1014.310,327.391,-148.956,170.222,52.120,160.192
C06151=1014.304,327.144,-148.922,170.215,52.125,160.192
C06152=1014.297,326.896,-148.888,170.207,52.130,160.192
C06153=1014.291,326.649,-148.854,170.200,52.135,160.191
C06154=1014.285,326.401,-148.820,170.194,52.140,160.191
C06155=1014.278,326.154,-148.786,170.187,52.144,160.191
C06156=1014.272,325.906,-148.752,170.179,52.150,160.191
C06157=1014.265,325.659,-148.718,170.172,52.155,160.191
C06158=1014.259,325.410,-148.685,170.165,52.160,160.191
C06159=1014.252,325.163,-148.651,170.159,52.165,160.190
C06160=1014.245,324.915,-148.617,170.151,52.170,160.190
C06161=1014.239,324.668,-148.585,170.144,52.175,160.190
C06162=1014.232,324.420,-148.551,170.138,52.180,160.190
C06163=1014.226,324.172,-148.518,170.130,52.186,160.190
C06164=1014.219,323.925,-148.484,170.124,52.191,160.190
C06165=1014.213,323.677,-148.451,170.117,52.196,160.190
C06166=1014.205,323.385,-148.411,170.108,52.202,160.189
C06167=1014.197,323.094,-148.373,170.100,52.208,160.189
C06168=1014.190,322.803,-148.333,170.093,52.214,160.189
C06169=1014.182,322.511,-148.293,170.084,52.220,160.189
C06170=1014.175,322.264,-148.260,170.078,52.225,160.189
C06171=1014.168,322.016,-148.227,170.071,52.230,160.189
C06172=1014.162,321.769,-148.194,170.063,52.236,160.189
C06173=1014.156,321.521,-148.161,170.057,52.241,160.189
C06174=1014.149,321.272,-148.127,170.050,52.246,160.189
C06175=1014.143,321.025,-148.094,170.042,52.252,160.188
C06176=1014.137,320.778,-148.061,170.036,52.257,160.188
C06177=1014.130,320.530,-148.029,170.029,52.262,160.188
C06178=1014.123,320.282,-147.995,170.023,52.267,160.188
C06179=1014.118,320.035,-147.961,170.016,52.272,160.188
C06180=1014.111,319.787,-147.929,170.009,52.278,160.188
C06181=1014.105,319.539,-147.896,170.002,52.283,160.188
C06182=1014.098,319.291,-147.863,169.996,52.289,160.188
C06183=1014.092,319.044,-147.830,169.989,52.294,160.188
C06184=1014.086,318.796,-147.796,169.981,52.299,160.188
C06185=1014.080,318.549,-147.763,169.975,52.305,160.188
C06186=1014.073,318.301,-147.730,169.968,52.310,160.188
C06187=1014.066,318.053,-147.697,169.962,52.316,160.188
C06188=1014.060,317.805,-147.665,169.954,52.321,160.188
C06189=1014.055,317.557,-147.631,169.948,52.327,160.188
C06190=1014.048,317.310,-147.599,169.941,52.332,160.188
C06191=1014.042,317.062,-147.566,169.935,52.337,160.188
C06192=1014.036,316.815,-147.533,169.928,52.342,160.188
C06193=1014.029,316.567,-147.500,169.921,52.349,160.188
C06194=1014.024,316.319,-147.467,169.915,52.354,160.188
C06195=1014.018,316.071,-147.434,169.908,52.359,160.188
C06196=1014.011,315.824,-147.402,169.902,52.365,160.188
C06197=1014.004,315.576,-147.368,169.894,52.370,160.187
C06198=1013.998,315.327,-147.336,169.888,52.376,160.187
C06199=1013.992,315.080,-147.304,169.882,52.382,160.188
C06200=1013.987,314.832,-147.270,169.875,52.387,160.187
C06201=1013.980,314.584,-147.238,169.869,52.392,160.188
C06202=1013.975,314.337,-147.205,169.861,52.398,160.188
C06203=1013.968,314.090,-147.172,169.855,52.403,160.187
C06204=1013.962,313.842,-147.140,169.848,52.409,160.187
C06205=1013.957,313.594,-147.107,169.842,52.415,160.188
C06206=1013.950,313.346,-147.074,169.836,52.420,160.188
C06207=1013.944,313.098,-147.042,169.829,52.426,160.188
C06208=1013.938,312.850,-147.010,169.822,52.431,160.187
C06209=1013.932,312.603,-146.977,169.815,52.437,160.188
C06210=1013.926,312.355,-146.944,169.809,52.443,160.188
C06211=1013.920,312.107,-146.911,169.803,52.449,160.188
C06212=1013.915,311.860,-146.879,169.797,52.454,160.188
C06213=1013.908,311.612,-146.846,169.789,52.460,160.188
C06214=1013.902,311.364,-146.814,169.783,52.465,160.188
C06215=1013.896,311.116,-146.782,169.776,52.471,160.188
C06216=1013.890,310.868,-146.750,169.770,52.477,160.188
C06217=1013.885,310.621,-146.717,169.764,52.482,160.188
C06218=1013.879,310.373,-146.684,169.758,52.488,160.188
C06219=1013.873,310.125,-146.652,169.750,52.494,160.188
C06220=1013.867,309.877,-146.619,169.744,52.500,160.188
C06221=1013.861,309.630,-146.587,169.738,52.505,160.188
C06222=1013.855,309.382,-146.555,169.732,52.511,160.188
C06223=1013.850,309.134,-146.522,169.725,52.517,160.188
C06224=1013.843,308.886,-146.491,169.718,52.523,160.188
C06225=1013.837,308.638,-146.459,169.712,52.529,160.189
C06226=1013.829,308.352,-146.422,169.705,52.535,160.189
C06227=1013.822,308.066,-146.386,169.697,52.542,160.189
C06228=1013.816,307.781,-146.349,169.689,52.550,160.189
C06229=1013.809,307.495,-146.312,169.682,52.556,160.189
C06230=1013.802,307.247,-146.281,169.677,52.563,160.189
C06231=1013.796,306.999,-146.249,169.669,52.569,160.189
C06232=1013.790,306.751,-146.218,169.663,52.575,160.189
C06233=1013.784,306.503,-146.186,169.657,52.581,160.190
C06234=1013.777,306.255,-146.154,169.651,52.587,160.190
C06235=1013.772,306.008,-146.123,169.644,52.593,160.190
C06236=1013.765,305.760,-146.091,169.638,52.599,160.190
C06237=1013.759,305.512,-146.059,169.632,52.605,160.190
C06238=1013.753,305.264,-146.028,169.625,52.612,160.190
C06239=1013.747,305.016,-145.996,169.619,52.617,160.190
C06240=1013.741,304.768,-145.966,169.612,52.623,160.190
C06241=1013.735,304.520,-145.934,169.606,52.629,160.191
C06242=1013.729,304.272,-145.902,169.599,52.635,160.191
C06243=1013.723,304.025,-145.871,169.593,52.642,160.191
C06244=1013.717,303.777,-145.839,169.587,52.647,160.191
C06245=1013.711,303.529,-145.808,169.580,52.654,160.191
C06246=1013.705,303.281,-145.776,169.574,52.660,160.191
C06247=1013.699,303.033,-145.745,169.568,52.666,160.192
C06248=1013.693,302.784,-145.714,169.562,52.673,160.192
C06249=1013.687,302.537,-145.683,169.555,52.679,160.192
C06250=1013.681,302.289,-145.651,169.549,52.685,160.192
C06251=1013.675,302.041,-145.621,169.543,52.691,160.192
C06252=1013.670,301.793,-145.588,169.537,52.697,160.193
C06253=1013.663,301.546,-145.557,169.530,52.704,160.193
C06254=1013.658,301.297,-145.526,169.524,52.710,160.193
C06255=1013.652,301.050,-145.495,169.518,52.716,160.193
C06256=1013.646,300.802,-145.463,169.513,52.723,160.194
C06257=1013.640,300.554,-145.433,169.505,52.729,160.194
C06258=1013.634,300.306,-145.401,169.500,52.735,160.194
C06259=1013.628,300.058,-145.370,169.494,52.741,160.194
C06260=1013.623,299.810,-145.339,169.488,52.748,160.194
C06261=1013.616,299.562,-145.308,169.481,52.754,160.194
C06262=1013.611,299.314,-145.276,169.475,52.760,160.195
C06263=1013.606,299.066,-145.245,169.469,52.767,160.195
C06264=1013.599,298.818,-145.215,169.462,52.774,160.195
C06265=1013.594,298.570,-145.183,169.456,52.780,160.195
C06266=1013.588,298.322,-145.153,169.450,52.786,160.196
C06267=1013.582,298.074,-145.121,169.444,52.792,160.196
C06268=1013.576,297.826,-145.090,169.438,52.799,160.196
C06269=1013.571,297.578,-145.059,169.432,52.805,160.196
C06270=1013.564,297.330,-145.028,169.426,52.812,160.197
C06271=1013.559,297.082,-144.997,169.420,52.818,160.197
C06272=1013.554,296.834,-144.967,169.413,52.825,160.197
C06273=1013.548,296.587,-144.935,169.408,52.831,160.197
C06274=1013.542,296.338,-144.904,169.401,52.837,160.197
C06275=1013.537,296.090,-144.873,169.395,52.844,160.198
C06276=1013.531,295.842,-144.843,169.389,52.850,160.198
C06277=1013.525,295.595,-144.811,169.383,52.857,160.198
C06278=1013.519,295.346,-144.780,169.377,52.863,160.199
C06279=1013.514,295.098,-144.750,169.371,52.870,160.199
C06280=1013.508,294.850,-144.719,169.364,52.876,160.199
C06281=1013.503,294.602,-144.688,169.359,52.883,160.199
C06282=1013.497,294.355,-144.657,169.353,52.889,160.200
C06283=1013.492,294.107,-144.626,169.347,52.896,160.200
C06284=1013.485,293.858,-144.596,169.341,52.903,160.200
C06285=1013.480,293.610,-144.565,169.335,52.910,160.201
C06286=1013.475,293.342,-144.532,169.328,52.916,160.201
C06287=1013.468,293.074,-144.498,169.322,52.924,160.201
C06288=1013.463,292.806,-144.465,169.315,52.931,160.201
C06289=1013.457,292.539,-144.432,169.309,52.938,160.202
C06290=1013.451,292.291,-144.401,169.303,52.945,160.202
C06291=1013.446,292.043,-144.371,169.297,52.951,160.202
C06292=1013.440,291.795,-144.341,169.292,52.958,160.203
C06293=1013.434,291.548,-144.310,169.285,52.965,160.203
C06294=1013.428,291.299,-144.281,169.279,52.971,160.203
C06295=1013.423,291.050,-144.249,169.273,52.978,160.204
C06296=1013.417,290.803,-144.219,169.267,52.985,160.204
C06297=1013.411,290.555,-144.189,169.261,52.992,160.204
C06298=1013.406,290.306,-144.159,169.256,52.999,160.205
C06299=1013.400,290.058,-144.129,169.249,53.006,160.205
C06300=1013.394,289.811,-144.098,169.243,53.012,160.205
C06301=1013.388,289.562,-144.069,169.238,53.019,160.206
C06302=1013.383,289.314,-144.038,169.231,53.026,160.206
C06303=1013.377,289.066,-144.009,169.226,53.033,160.207
C06304=1013.371,288.818,-143.978,169.220,53.040,160.207
C06305=1013.365,288.570,-143.948,169.214,53.047,160.207
C06306=1013.360,288.322,-143.918,169.208,53.054,160.208
C06307=1013.354,288.074,-143.888,169.202,53.061,160.208
C06308=1013.349,287.826,-143.858,169.196,53.067,160.208
C06309=1013.343,287.578,-143.828,169.191,53.075,160.209
C06310=1013.338,287.330,-143.799,169.184,53.081,160.209
C06311=1013.332,287.082,-143.769,169.178,53.089,160.209
C06312=1013.327,286.834,-143.739,169.173,53.096,160.210
C06313=1013.321,286.585,-143.709,169.166,53.103,160.210
C06314=1013.315,286.338,-143.679,169.161,53.110,160.211
C06315=1013.310,286.089,-143.649,169.155,53.116,160.211
C06316=1013.304,285.841,-143.620,169.149,53.124,160.211
C06317=1013.298,285.593,-143.589,169.144,53.131,160.212
C06318=1013.293,285.344,-143.560,169.137,53.138,160.212
C06319=1013.288,285.097,-143.530,169.132,53.145,160.213
C06320=1013.282,284.849,-143.500,169.126,53.152,160.213
C06321=1013.277,284.600,-143.470,169.120,53.159,160.214
C06322=1013.271,284.352,-143.441,169.114,53.166,160.214
C06323=1013.266,284.103,-143.411,169.109,53.173,160.214
C06324=1013.259,283.856,-143.381,169.102,53.181,160.215
C06325=1013.254,283.608,-143.352,169.097,53.188,160.215
C06326=1013.249,283.360,-143.322,169.091,53.195,160.216
C06327=1013.243,283.111,-143.293,169.085,53.202,160.216
C06328=1013.237,282.863,-143.264,169.079,53.209,160.216
C06329=1013.231,282.615,-143.234,169.073,53.216,160.217
C06330=1013.226,282.367,-143.205,169.068,53.224,160.217
C06331=1013.220,282.119,-143.176,169.062,53.231,160.218
C06332=1013.215,281.870,-143.146,169.057,53.238,160.218
C06333=1013.209,281.622,-143.117,169.050,53.246,160.219
C06334=1013.204,281.374,-143.087,169.045,53.253,160.219
C06335=1013.198,281.126,-143.058,169.039,53.261,160.220
C06336=1013.193,280.878,-143.029,169.033,53.268,160.220
C06337=1013.188,280.630,-142.999,169.028,53.275,160.221
C06338=1013.181,280.382,-142.970,169.022,53.282,160.221
C06339=1013.176,280.133,-142.941,169.016,53.290,160.221
C06340=1013.171,279.884,-142.912,169.010,53.297,160.222
C06341=1013.166,279.637,-142.882,169.005,53.304,160.222
C06342=1013.159,279.388,-142.853,168.998,53.312,160.223
C06343=1013.154,279.140,-142.824,168.993,53.319,160.223
C06344=1013.149,278.892,-142.795,168.988,53.326,160.224
C06345=1013.143,278.643,-142.766,168.982,53.334,160.224
C06346=1013.138,278.388,-142.736,168.976,53.342,160.225
C06347=1013.132,278.133,-142.706,168.970,53.349,160.225
C06348=1013.127,277.877,-142.675,168.964,53.357,160.226
C06349=1013.121,277.622,-142.645,168.958,53.365,160.226
C06350=1013.116,277.373,-142.617,168.953,53.372,160.227
C06351=1013.111,277.125,-142.587,168.948,53.379,160.227
C06352=1013.104,276.877,-142.558,168.941,53.387,160.228
C06353=1013.100,276.628,-142.530,168.936,53.394,160.228
C06354=1013.094,276.380,-142.500,168.930,53.402,160.229
C06355=1013.089,276.132,-142.471,168.925,53.410,160.229
C06356=1013.083,275.883,-142.442,168.919,53.417,160.230
C06357=1013.079,275.636,-142.413,168.913,53.424,160.230
C06358=1013.072,275.387,-142.384,168.908,53.433,160.231
C06359=1013.067,275.139,-142.356,168.902,53.440,160.231
C06360=1013.062,274.890,-142.327,168.896,53.447,160.232
C06361=1013.056,274.643,-142.299,168.891,53.455,160.233
C06362=1013.051,274.394,-142.270,168.885,53.463,160.233
C06363=1013.045,274.146,-142.241,168.880,53.470,160.233
C06364=1013.040,273.897,-142.212,168.874,53.478,160.234
C06365=1013.034,273.650,-142.183,168.869,53.485,160.235
C06366=1013.029,273.401,-142.154,168.863,53.494,160.235
C06367=1013.024,273.153,-142.127,168.858,53.501,160.236
C06368=1013.018,272.904,-142.097,168.852,53.509,160.236
C06369=1013.013,272.656,-142.069,168.846,53.516,160.237
C06370=1013.008,272.408,-142.041,168.840,53.524,160.237
C06371=1013.002,272.160,-142.011,168.835,53.532,160.238
C06372=1012.997,271.912,-141.983,168.829,53.539,160.238
C06373=1012.992,271.663,-141.954,168.824,53.547,160.239
C06374=1012.983,271.319,-141.915,168.816,53.558,160.240
C06375=1012.977,270.975,-141.876,168.808,53.569,160.241
C06376=1012.970,270.631,-141.836,168.801,53.580,160.241
C06377=1012.962,270.286,-141.797,168.793,53.591,160.242
C06378=1012.768,273.436,-142.522,168.831,53.604,160.253
C06379=1012.773,273.740,-142.558,168.838,53.594,160.253
C06380=1012.780,274.045,-142.593,168.844,53.585,160.252
C06381=1012.787,274.350,-142.628,168.852,53.575,160.251
C06382=1012.794,274.654,-142.663,168.858,53.566,160.250
C06383=1012.799,274.903,-142.692,168.864,53.558,160.250
C06384=1012.805,275.151,-142.721,168.871,53.550,160.250
C06385=1012.810,275.399,-142.749,168.875,53.543,160.249
C06386=1012.816,275.647,-142.778,168.882,53.535,160.249
C06387=1012.821,275.896,-142.807,168.887,53.528,160.248
C06388=1012.827,276.144,-142.836,168.893,53.519,160.247
C06389=1012.831,276.392,-142.864,168.898,53.512,160.247
C06390=1012.837,276.641,-142.894,168.904,53.505,160.247
C06391=1012.842,276.888,-142.923,168.910,53.497,160.246
C06392=1012.848,277.137,-142.952,168.915,53.489,160.245
C06393=1012.853,277.385,-142.981,168.921,53.482,160.245
C06394=1012.858,277.633,-143.011,168.927,53.474,160.245
C06395=1012.864,277.892,-143.040,168.932,53.467,160.244
C06396=1012.869,278.148,-143.070,168.938,53.459,160.243
C06397=1012.875,278.406,-143.100,168.944,53.451,160.243
C06398=1012.880,278.664,-143.131,168.950,53.443,160.242
C06399=1012.886,278.912,-143.160,168.955,53.436,160.242
C06400=1012.892,279.161,-143.189,168.962,53.428,160.241
C06401=1012.896,279.409,-143.218,168.967,53.421,160.241
C06402=1012.902,279.658,-143.248,168.973,53.414,160.241
C06403=1012.908,279.905,-143.277,168.979,53.406,160.240
C06404=1012.913,280.154,-143.306,168.985,53.399,160.240
C06405=1012.918,280.403,-143.335,168.990,53.392,160.239
C06406=1012.924,280.650,-143.364,168.996,53.384,160.239
C06407=1012.930,280.898,-143.393,169.002,53.377,160.238
C06408=1012.935,281.147,-143.423,169.008,53.369,160.238
C06409=1012.940,281.395,-143.452,169.013,53.362,160.237
C06410=1012.946,281.643,-143.481,169.020,53.355,160.237
C06411=1012.952,281.891,-143.511,169.025,53.347,160.236
C06412=1012.957,282.140,-143.541,169.031,53.340,160.236
C06413=1012.963,282.387,-143.569,169.036,53.333,160.235
C06414=1012.968,282.636,-143.598,169.043,53.325,160.235
C06415=1012.974,282.885,-143.628,169.048,53.318,160.235
C06416=1012.980,283.133,-143.657,169.054,53.310,160.234
C06417=1012.985,283.380,-143.686,169.060,53.303,160.234
C06418=1012.990,283.629,-143.716,169.066,53.296,160.234
C06419=1012.996,283.877,-143.746,169.072,53.289,160.233
C06420=1013.002,284.125,-143.775,169.077,53.282,160.232
C06421=1013.007,284.373,-143.804,169.083,53.274,160.232
C06422=1013.013,284.621,-143.834,169.089,53.267,160.232
C06423=1013.018,284.869,-143.864,169.095,53.260,160.231
C06424=1013.024,285.117,-143.894,169.101,53.253,160.231
C06425=1013.030,285.366,-143.924,169.107,53.246,160.230
C06426=1013.034,285.613,-143.953,169.112,53.239,160.230
C06427=1013.040,285.862,-143.983,169.118,53.232,160.230
C06428=1013.046,286.110,-144.013,169.124,53.225,160.229
C06429=1013.051,286.358,-144.043,169.130,53.217,160.229
C06430=1013.057,286.607,-144.072,169.136,53.210,160.229
C06431=1013.063,286.854,-144.103,169.142,53.203,160.228
C06432=1013.068,287.103,-144.132,169.148,53.196,160.228
C06433=1013.073,287.351,-144.162,169.154,53.189,160.227
C06434=1013.079,287.598,-144.192,169.159,53.182,160.227
C06435=1013.084,287.847,-144.221,169.166,53.175,160.227
C06436=1013.090,288.095,-144.252,169.171,53.168,160.226
C06437=1013.096,288.343,-144.281,169.177,53.161,160.226
C06438=1013.102,288.591,-144.312,169.183,53.154,160.225
C06439=1013.107,288.839,-144.341,169.189,53.147,160.225
C06440=1013.113,289.087,-144.372,169.195,53.140,160.225
C06441=1013.118,289.336,-144.401,169.201,53.133,160.224
C06442=1013.124,289.584,-144.432,169.207,53.126,160.224
C06443=1013.130,289.832,-144.461,169.213,53.119,160.224
C06444=1013.136,290.080,-144.492,169.219,53.113,160.223
C06445=1013.141,290.328,-144.521,169.225,53.105,160.223
C06446=1013.147,290.576,-144.552,169.231,53.099,160.223
C06447=1013.153,290.824,-144.582,169.237,53.092,160.222
C06448=1013.158,291.072,-144.613,169.243,53.085,160.222
C06449=1013.163,291.320,-144.643,169.248,53.078,160.222
C06450=1013.169,291.568,-144.673,169.255,53.071,160.221
C06451=1013.175,291.816,-144.703,169.261,53.064,160.221
C06452=1013.181,292.064,-144.734,169.267,53.057,160.221
C06453=1013.186,292.312,-144.763,169.273,53.051,160.220
C06454=1013.191,292.560,-144.794,169.278,53.044,160.220
C06455=1013.198,292.830,-144.828,169.285,53.037,160.220
C06456=1013.204,293.100,-144.861,169.292,53.030,160.219
C06457=1013.209,293.370,-144.895,169.298,53.022,160.219
C06458=1013.215,293.641,-144.928,169.305,53.015,160.219
C06459=1013.221,293.889,-144.958,169.311,53.008,160.219
C06460=1013.226,294.136,-144.990,169.317,53.002,160.218
C06461=1013.232,294.384,-145.020,169.323,52.995,160.218
C06462=1013.238,294.633,-145.052,169.329,52.988,160.218
C06463=1013.243,294.881,-145.082,169.335,52.982,160.217
C06464=1013.249,295.129,-145.113,169.341,52.975,160.217
C06465=1013.254,295.376,-145.143,169.348,52.968,160.217
C06466=1013.259,295.625,-145.174,169.354,52.962,160.217
C06467=1013.265,295.872,-145.204,169.359,52.955,160.216
C06468=1013.271,296.121,-145.237,169.366,52.949,160.216
C06469=1013.277,296.368,-145.267,169.372,52.942,160.216
C06470=1013.282,296.617,-145.298,169.378,52.936,160.215
C06471=1013.288,296.864,-145.328,169.384,52.929,160.215
C06472=1013.293,297.112,-145.360,169.390,52.923,160.215
C06473=1013.300,297.360,-145.391,169.396,52.916,160.215
C06474=1013.305,297.609,-145.421,169.403,52.909,160.214
C06475=1013.311,297.856,-145.452,169.409,52.904,160.214
C06476=1013.316,298.104,-145.483,169.415,52.897,160.214
C06477=1013.322,298.352,-145.514,169.421,52.891,160.214
C06478=1013.328,298.601,-145.545,169.427,52.884,160.214
C06479=1013.334,298.848,-145.576,169.433,52.877,160.213
C06480=1013.339,299.097,-145.608,169.439,52.871,160.213
C06481=1013.346,299.344,-145.639,169.446,52.864,160.213
C06482=1013.351,299.592,-145.670,169.452,52.859,160.213
C06483=1013.357,299.840,-145.702,169.458,52.852,160.212
C06484=1013.362,300.088,-145.732,169.465,52.845,160.212
C06485=1013.367,300.336,-145.763,169.470,52.839,160.212
C06486=1013.374,300.584,-145.794,169.476,52.832,160.212
C06487=1013.379,300.832,-145.825,169.484,52.826,160.212
C06488=1013.386,301.080,-145.857,169.489,52.820,160.211
C06489=1013.391,301.328,-145.888,169.495,52.814,160.211
C06490=1013.397,301.575,-145.919,169.502,52.807,160.211
C06491=1013.403,301.824,-145.951,169.508,52.801,160.211
C06492=1013.409,302.071,-145.981,169.514,52.795,160.211
C06493=1013.415,302.320,-146.013,169.521,52.788,160.211
C06494=1013.421,302.567,-146.043,169.527,52.782,160.210
C06495=1013.427,302.816,-146.075,169.533,52.776,160.210
C06496=1013.433,303.063,-146.107,169.540,52.770,160.210
C06497=1013.439,303.312,-146.138,169.546,52.763,160.210
C06498=1013.445,303.559,-146.169,169.552,52.757,160.209
C06499=1013.451,303.807,-146.201,169.559,52.751,160.209
C06500=1013.457,304.054,-146.232,169.565,52.744,160.209
C06501=1013.463,304.303,-146.263,169.571,52.739,160.209
C06502=1013.469,304.550,-146.294,169.578,52.732,160.209
C06503=1013.475,304.799,-146.326,169.584,52.726,160.209
C06504=1013.481,305.046,-146.357,169.590,52.720,160.209
C06505=1013.486,305.295,-146.389,169.597,52.714,160.209
C06506=1013.492,305.543,-146.421,169.603,52.707,160.208
C06507=1013.499,305.790,-146.452,169.609,52.701,160.208
C06508=1013.505,306.038,-146.484,169.616,52.695,160.208
C06509=1013.511,306.286,-146.515,169.622,52.689,160.208
C06510=1013.517,306.534,-146.547,169.628,52.683,160.208
C06511=1013.523,306.782,-146.578,169.635,52.676,160.208
C06512=1013.529,307.030,-146.610,169.642,52.671,160.208
C06513=1013.535,307.277,-146.642,169.647,52.664,160.207
C06514=1013.541,307.526,-146.673,169.655,52.658,160.207
C06515=1013.549,307.814,-146.710,169.661,52.651,160.207
C06516=1013.556,308.102,-146.747,169.669,52.644,160.207
C06517=1013.564,308.390,-146.784,169.677,52.637,160.207
C06518=1013.570,308.679,-146.820,169.685,52.630,160.207
C06519=1013.576,308.926,-146.852,169.691,52.624,160.206
C06520=1013.583,309.173,-146.884,169.697,52.618,160.206
C06521=1013.588,309.421,-146.916,169.703,52.612,160.206
C06522=1013.594,309.669,-146.949,169.710,52.606,160.206
C06523=1013.600,309.917,-146.981,169.717,52.600,160.206
C06524=1013.606,310.165,-147.013,169.723,52.595,160.206
C06525=1013.611,310.412,-147.045,169.729,52.589,160.206
C06526=1013.617,310.660,-147.077,169.736,52.583,160.206
C06527=1013.624,310.908,-147.110,169.743,52.577,160.206
C06528=1013.629,311.156,-147.143,169.749,52.572,160.206
C06529=1013.635,311.403,-147.175,169.755,52.566,160.206
C06530=1013.641,311.651,-147.208,169.763,52.560,160.206
C06531=1013.647,311.899,-147.240,169.769,52.554,160.206
C06532=1013.653,312.147,-147.273,169.775,52.548,160.206
C06533=1013.659,312.395,-147.305,169.781,52.543,160.206
C06534=1013.664,312.642,-147.338,169.789,52.537,160.206
C06535=1013.670,312.890,-147.370,169.795,52.532,160.206
C06536=1013.676,313.138,-147.402,169.802,52.526,160.206
C06537=1013.683,313.386,-147.435,169.808,52.520,160.206
C06538=1013.689,313.633,-147.468,169.815,52.514,160.206
C06539=1013.694,313.882,-147.501,169.821,52.508,160.206
C06540=1013.701,314.129,-147.533,169.828,52.503,160.206
C06541=1013.707,314.377,-147.566,169.834,52.498,160.206
C06542=1013.713,314.624,-147.599,169.842,52.492,160.206
C06543=1013.719,314.872,-147.631,169.848,52.486,160.205
C06544=1013.725,315.120,-147.663,169.854,52.480,160.205
C06545=1013.730,315.367,-147.696,169.861,52.475,160.206
C06546=1013.737,315.615,-147.729,169.868,52.469,160.206
C06547=1013.743,315.863,-147.762,169.874,52.463,160.205
C06548=1013.749,316.110,-147.795,169.881,52.458,160.206
C06549=1013.756,316.358,-147.827,169.888,52.452,160.206
C06550=1013.762,316.606,-147.861,169.895,52.447,160.206
C06551=1013.768,316.855,-147.893,169.901,52.442,160.206
C06552=1013.774,317.102,-147.926,169.908,52.436,160.206
C06553=1013.780,317.350,-147.959,169.915,52.431,160.206
C06554=1013.787,317.597,-147.991,169.922,52.425,160.206
C06555=1013.792,317.845,-148.025,169.928,52.419,160.206
C06556=1013.798,318.093,-148.058,169.935,52.414,160.206
C06557=1013.805,318.340,-148.090,169.942,52.408,160.206
C06558=1013.811,318.588,-148.123,169.948,52.403,160.206
C06559=1013.818,318.835,-148.156,169.955,52.397,160.206
C06560=1013.824,319.083,-148.190,169.962,52.392,160.206
C06561=1013.830,319.331,-148.223,169.969,52.386,160.206
C06562=1013.836,319.579,-148.256,169.975,52.381,160.206
C06563=1013.843,319.826,-148.288,169.983,52.375,160.206
C06564=1013.849,320.074,-148.321,169.989,52.370,160.206
C06565=1013.856,320.322,-148.354,169.996,52.365,160.206
C06566=1013.862,320.570,-148.388,170.003,52.359,160.206
C06567=1013.868,320.817,-148.421,170.010,52.354,160.206
C06568=1013.874,321.065,-148.454,170.016,52.349,160.206
C06569=1013.881,321.313,-148.487,170.024,52.343,160.207
C06570=1013.888,321.560,-148.520,170.031,52.338,160.207
C06571=1013.893,321.808,-148.554,170.037,52.333,160.207
C06572=1013.900,322.056,-148.587,170.045,52.327,160.207
C06573=1013.906,322.304,-148.620,170.051,52.322,160.207
C06574=1013.913,322.551,-148.653,170.058,52.317,160.207
C06575=1013.920,322.845,-148.692,170.066,52.311,160.207
C06576=1013.928,323.138,-148.732,170.075,52.304,160.207
C06577=1013.936,323.432,-148.772,170.083,52.298,160.207
C06578=1013.944,323.726,-148.811,170.091,52.291,160.208
C06579=1013.951,323.973,-148.844,170.098,52.286,160.208
C06580=1013.956,324.221,-148.878,170.105,52.281,160.208
C06581=1013.963,324.469,-148.911,170.112,52.276,160.208
C06582=1013.970,324.716,-148.944,170.119,52.271,160.208
C06583=1013.977,324.964,-148.978,170.125,52.265,160.208
C06584=1013.983,325.211,-149.011,170.133,52.260,160.208
C06585=1013.990,325.459,-149.045,170.140,52.255,160.208
C06586=1013.996,325.706,-149.079,170.148,52.250,160.209
C06587=1014.003,325.955,-149.112,170.154,52.245,160.209
C06588=1014.009,326.202,-149.146,170.161,52.240,160.209
C06589=1014.016,326.450,-149.180,170.168,52.235,160.209
C06590=1014.022,326.697,-149.214,170.176,52.230,160.209
C06591=1014.029,326.945,-149.248,170.183,52.225,160.210
C06592=1014.034,327.192,-149.282,170.189,52.220,160.210
C06593=1014.042,327.440,-149.316,170.197,52.215,160.210
C06594=1014.048,327.688,-149.350,170.204,52.210,160.210
C06595=1014.054,327.935,-149.384,170.210,52.205,160.210
C06596=1014.061,328.183,-149.418,170.219,52.200,160.211
C06597=1014.067,328.430,-149.452,170.225,52.195,160.211
C06598=1014.074,328.678,-149.487,170.232,52.190,160.211
C06599=1014.080,328.925,-149.520,170.239,52.185,160.211
C06600=1014.087,329.173,-149.555,170.247,52.180,160.211
C06601=1014.093,329.421,-149.589,170.254,52.175,160.211
C06602=1014.100,329.668,-149.622,170.260,52.170,160.212
C06603=1014.106,329.916,-149.657,170.268,52.166,160.212
C06604=1014.113,330.164,-149.691,170.275,52.161,160.212
C06605=1014.120,330.412,-149.725,170.282,52.156,160.212
C06606=1014.126,330.658,-149.760,170.290,52.151,160.213
C06607=1014.132,330.906,-149.794,170.297,52.146,160.213
C06608=1014.140,331.154,-149.828,170.303,52.141,160.213
C06609=1014.145,331.401,-149.862,170.312,52.136,160.213
C06610=1014.152,331.649,-149.897,170.318,52.131,160.213
C06611=1014.159,331.896,-149.931,170.325,52.127,160.214
C06612=1014.166,332.144,-149.966,170.333,52.122,160.214
C06613=1014.173,332.392,-150.001,170.340,52.117,160.214
C06614=1014.179,332.639,-150.035,170.347,52.112,160.214
C06615=1014.185,332.886,-150.070,170.355,52.108,160.215
C06616=1014.192,333.134,-150.104,170.362,52.103,160.215
C06617=1014.199,333.382,-150.139,170.369,52.098,160.215
C06618=1014.206,333.629,-150.173,170.377,52.094,160.216
C06619=1014.212,333.876,-150.208,170.384,52.089,160.216
C06620=1014.218,334.124,-150.242,170.391,52.084,160.216
C06621=1014.225,334.371,-150.278,170.399,52.080,160.217
C06622=1014.232,334.619,-150.313,170.406,52.075,160.217
C06623=1014.238,334.867,-150.347,170.413,52.070,160.217
C06624=1014.245,335.114,-150.382,170.421,52.066,160.218
C06625=1014.252,335.361,-150.417,170.428,52.061,160.218
C06626=1014.258,335.609,-150.452,170.435,52.057,160.218
C06627=1014.265,335.857,-150.487,170.443,52.052,160.218
C06628=1014.272,336.104,-150.522,170.450,52.047,160.219
C06629=1014.279,336.352,-150.557,170.458,52.043,160.219
C06630=1014.286,336.599,-150.591,170.466,52.038,160.220
C06631=1014.293,336.847,-150.626,170.473,52.034,160.220
C06632=1014.299,337.094,-150.661,170.481,52.029,160.220
C06633=1014.306,337.341,-150.696,170.488,52.025,160.221
C06634=1014.313,337.589,-150.732,170.495,52.021,160.221
C06635=1014.321,337.878,-150.773,170.504,52.015,160.221
C06636=1014.329,338.168,-150.814,170.513,52.010,160.222
C06637=1014.336,338.456,-150.855,170.522,52.004,160.222
C06638=1014.344,338.746,-150.896,170.531,51.999,160.223
C06639=1014.351,338.994,-150.931,170.538,51.995,160.223
C06640=1014.358,339.241,-150.966,170.545,51.990,160.223
C06641=1014.365,339.488,-151.001,170.553,51.986,160.224
C06642=1014.372,339.736,-151.038,170.561,51.982,160.224
C06643=1014.378,339.983,-151.073,170.569,51.977,160.225
C06644=1014.385,340.231,-151.109,170.576,51.973,160.225
C06645=1014.392,340.478,-151.144,170.583,51.969,160.225
C06646=1014.399,340.725,-151.180,170.591,51.964,160.226
C06647=1014.406,340.973,-151.215,170.599,51.960,160.226
C06648=1014.412,341.221,-151.251,170.607,51.956,160.227
C06649=1014.420,341.467,-151.287,170.614,51.951,160.227
C06650=1014.426,341.715,-151.322,170.621,51.947,160.227
C06651=1014.434,341.963,-151.357,170.630,51.943,160.228
C06652=1014.441,342.210,-151.393,170.637,51.939,160.228
C06653=1014.447,342.457,-151.429,170.645,51.934,160.229
C06654=1014.454,342.704,-151.465,170.653,51.931,160.229
C06655=1014.461,342.952,-151.500,170.660,51.926,160.230
C06656=1014.468,343.199,-151.536,170.669,51.922,160.230
C06657=1014.474,343.446,-151.572,170.676,51.918,160.231
C06658=1014.482,343.694,-151.608,170.684,51.913,160.231
C06659=1014.489,343.941,-151.643,170.691,51.910,160.232
C06660=1014.496,344.188,-151.679,170.700,51.905,160.232
C06661=1014.503,344.436,-151.716,170.707,51.901,160.233
C06662=1014.510,344.683,-151.751,170.714,51.897,160.233
C06663=1014.517,344.931,-151.787,170.723,51.893,160.233
C06664=1014.524,345.178,-151.824,170.730,51.889,160.234
C06665=1014.531,345.426,-151.859,170.739,51.885,160.234
C06666=1014.538,345.672,-151.895,170.746,51.881,160.235
C06667=1014.546,345.920,-151.931,170.754,51.876,160.235
C06668=1014.552,346.167,-151.968,170.762,51.873,160.236
C06669=1014.560,346.414,-152.004,170.770,51.869,160.237
C06670=1014.567,346.661,-152.040,170.778,51.864,160.237
C06671=1014.574,346.909,-152.076,170.786,51.860,160.238
C06672=1014.581,347.156,-152.112,170.794,51.857,160.238
C06673=1014.588,347.403,-152.149,170.802,51.853,160.239
C06674=1014.595,347.650,-152.185,170.809,51.848,160.239
C06675=1014.602,347.898,-152.222,170.818,51.844,160.240
C06676=1014.609,348.145,-152.258,170.826,51.841,160.240
C06677=1014.616,348.392,-152.294,170.834,51.837,160.241
C06678=1014.623,348.640,-152.331,170.842,51.833,160.241
C06679=1014.630,348.887,-152.367,170.850,51.829,160.242
C06680=1014.637,349.134,-152.403,170.858,51.825,160.243
C06681=1014.644,349.381,-152.440,170.866,51.821,160.243
C06682=1014.652,349.628,-152.477,170.874,51.818,160.244
C06683=1014.659,349.876,-152.514,170.883,51.813,160.244
C06684=1014.666,350.123,-152.549,170.890,51.810,160.245
C06685=1014.673,350.370,-152.587,170.899,51.806,160.246
C06686=1014.680,350.618,-152.624,170.906,51.802,160.246
C06687=1014.688,350.865,-152.660,170.915,51.798,160.247
C06688=1014.694,351.111,-152.697,170.922,51.794,160.247
C06689=1014.702,351.359,-152.733,170.931,51.790,160.248
C06690=1014.709,351.606,-152.771,170.939,51.787,160.248
C06691=1014.717,351.853,-152.807,170.947,51.783,160.249
C06692=1014.724,352.101,-152.845,170.955,51.779,160.250
C06693=1014.731,352.347,-152.880,170.963,51.775,160.250
C06694=1014.738,352.594,-152.918,170.972,51.772,160.251
C06695=1014.747,352.881,-152.960,170.981,51.768,160.252
C06696=1014.756,353.168,-153.003,170.990,51.763,160.252
C06697=1014.764,353.455,-153.046,171.000,51.759,160.253
C06698=1014.773,353.742,-153.089,171.010,51.755,160.254
C06699=1014.780,353.989,-153.126,171.019,51.751,160.255
C06700=1014.788,354.236,-153.164,171.026,51.748,160.255
C06701=1014.794,354.482,-153.201,171.035,51.743,160.256
C06702=1014.801,354.730,-153.238,171.044,51.740,160.257
C06703=1014.809,354.977,-153.275,171.051,51.736,160.257
C06704=1014.817,355.224,-153.312,171.060,51.733,160.258
C06705=1014.824,355.471,-153.350,171.068,51.729,160.259
C06706=1014.831,355.718,-153.387,171.077,51.726,160.259
C06707=1014.839,355.965,-153.424,171.085,51.722,160.260
C06708=1014.846,356.212,-153.462,171.093,51.719,160.261
C06709=1014.854,356.459,-153.499,171.102,51.715,160.261
C06710=1014.861,356.706,-153.536,171.111,51.712,160.262
C06711=1014.869,356.954,-153.574,171.119,51.709,160.263
C06712=1014.877,357.201,-153.612,171.127,51.705,160.264
C06713=1014.884,357.448,-153.649,171.136,51.701,160.264
C06714=1014.891,357.696,-153.687,171.144,51.698,160.265
C06715=1014.899,357.942,-153.724,171.153,51.694,160.266
C06716=1014.907,358.189,-153.762,171.162,51.691,160.267
C06717=1014.914,358.436,-153.799,171.170,51.688,160.267
C06718=1014.922,358.684,-153.837,171.178,51.684,160.268
C06719=1014.929,358.930,-153.875,171.187,51.680,160.269
C06720=1014.936,359.177,-153.913,171.195,51.677,160.270
C06721=1014.944,359.425,-153.950,171.204,51.674,160.271
C06722=1014.951,359.671,-153.989,171.213,51.671,160.271
C06723=1014.959,359.918,-154.026,171.221,51.668,160.272
C06724=1014.967,360.165,-154.065,171.230,51.664,160.273
C06725=1014.974,360.413,-154.102,171.239,51.661,160.274
C06726=1014.981,360.659,-154.141,171.247,51.658,160.275
C06727=1014.989,360.906,-154.179,171.256,51.655,160.275
C06728=1014.997,361.153,-154.217,171.265,51.651,160.276
C06729=1015.004,361.400,-154.255,171.273,51.648,160.277
C06730=1015.012,361.647,-154.293,171.282,51.645,160.278
C06731=1015.020,361.894,-154.331,171.291,51.641,160.279
C06732=1015.027,362.141,-154.369,171.300,51.638,160.279
C06733=1015.036,362.388,-154.408,171.308,51.635,160.280
C06734=1015.043,362.635,-154.446,171.317,51.632,160.281
C06735=1015.050,362.882,-154.484,171.327,51.629,160.282
C06736=1015.058,363.129,-154.523,171.336,51.625,160.283
C06737=1015.065,363.376,-154.561,171.344,51.622,160.284
C06738=1015.073,363.623,-154.600,171.353,51.619,160.284
C06739=1015.081,363.870,-154.638,171.362,51.616,160.286
C06740=1015.089,364.117,-154.677,171.371,51.613,160.286
C06741=1015.097,364.363,-154.715,171.380,51.610,160.287
C06742=1015.105,364.610,-154.754,171.388,51.607,160.288
C06743=1015.112,364.857,-154.792,171.397,51.604,160.289
C06744=1015.121,365.104,-154.830,171.406,51.600,160.290
C06745=1015.128,365.351,-154.869,171.416,51.598,160.291
C06746=1015.136,365.598,-154.907,171.425,51.594,160.292
C06747=1015.144,365.845,-154.946,171.434,51.592,160.293
C06748=1015.152,366.092,-154.984,171.442,51.589,160.294
C06749=1015.160,366.339,-155.023,171.451,51.585,160.294
C06750=1015.168,366.585,-155.062,171.460,51.582,160.295
C06751=1015.176,366.832,-155.100,171.470,51.580,160.296
C06752=1015.184,367.079,-155.139,171.479,51.576,160.297
C06753=1015.191,367.326,-155.178,171.488,51.574,160.298
C06754=1015.199,367.573,-155.217,171.497,51.570,160.299
C06755=1015.208,367.867,-155.263,171.508,51.567,160.300
C06756=1015.218,368.161,-155.310,171.519,51.564,160.302
C06757=1015.228,368.456,-155.357,171.529,51.560,160.303
C06758=1015.237,368.750,-155.403,171.541,51.557,160.304
C06759=1015.245,368.997,-155.443,171.550,51.554,160.305
C06760=1015.253,369.243,-155.482,171.559,51.551,160.306
C06761=1015.261,369.490,-155.521,171.569,51.549,160.307
C06762=1015.268,369.737,-155.561,171.578,51.545,160.308
C06763=1015.277,369.984,-155.600,171.587,51.543,160.309
C06764=1015.285,370.231,-155.639,171.596,51.540,160.310
C06765=1015.293,370.478,-155.679,171.605,51.537,160.311
C06766=1015.301,370.724,-155.718,171.614,51.535,160.312
C06767=1015.308,370.971,-155.758,171.624,51.532,160.313
C06768=1015.317,371.217,-155.797,171.633,51.529,160.314
C06769=1015.325,371.464,-155.836,171.643,51.526,160.315
C06770=1015.333,371.711,-155.876,171.652,51.524,160.316
C06771=1015.341,371.957,-155.915,171.661,51.521,160.317
C06772=1015.350,372.204,-155.955,171.671,51.519,160.318
C06773=1015.358,372.451,-155.995,171.681,51.516,160.320
C06774=1015.366,372.697,-156.034,171.690,51.513,160.321
C06775=1015.374,372.944,-156.074,171.699,51.510,160.322
C06776=1015.382,373.191,-156.113,171.709,51.508,160.323
C06777=1015.391,373.438,-156.153,171.719,51.505,160.324
C06778=1015.398,373.684,-156.193,171.729,51.502,160.325
C06779=1015.407,373.931,-156.232,171.738,51.500,160.326
C06780=1015.415,374.179,-156.272,171.748,51.497,160.327
C06781=1015.424,374.425,-156.312,171.758,51.495,160.328
C06782=1015.432,374.671,-156.352,171.767,51.492,160.329
C06783=1015.440,374.918,-156.391,171.776,51.489,160.330
C06784=1015.449,375.164,-156.431,171.786,51.487,160.332
C06785=1015.458,375.411,-156.471,171.795,51.484,160.333
C06786=1015.466,375.658,-156.511,171.805,51.482,160.334
C06787=1015.474,375.905,-156.552,171.816,51.479,160.335
C06788=1015.482,376.151,-156.592,171.825,51.477,160.336
C06789=1015.490,376.397,-156.632,171.835,51.475,160.338
C06790=1015.499,376.644,-156.673,171.845,51.472,160.339
C06791=1015.507,376.891,-156.713,171.854,51.470,160.340
C06792=1015.515,377.138,-156.753,171.864,51.468,160.341
C06793=1015.523,377.384,-156.793,171.874,51.465,160.342
C06794=1015.532,377.631,-156.834,171.884,51.463,160.344
C06795=1015.540,377.877,-156.875,171.894,51.460,160.345
C06796=1015.549,378.123,-156.915,171.904,51.458,160.346
C06797=1015.557,378.370,-156.955,171.913,51.456,160.347
C06798=1015.565,378.617,-156.996,171.923,51.453,160.348
C06799=1015.574,378.864,-157.037,171.934,51.451,160.350
C06800=1015.583,379.110,-157.077,171.944,51.449,160.351
C06801=1015.591,379.356,-157.118,171.954,51.447,160.352
C06802=1015.599,379.603,-157.159,171.963,51.444,160.354
C06803=1015.607,379.849,-157.199,171.974,51.442,160.355
C06804=1015.617,380.096,-157.240,171.984,51.440,160.356
C06805=1015.625,380.342,-157.281,171.994,51.438,160.357
C06806=1015.634,380.589,-157.322,172.004,51.435,160.359
C06807=1015.642,380.835,-157.362,172.014,51.433,160.360
C06808=1015.651,381.082,-157.403,172.024,51.431,160.361
C06809=1015.660,381.329,-157.444,172.034,51.429,160.363
C06810=1015.668,381.574,-157.485,172.045,51.426,160.364
C06811=1015.677,381.821,-157.526,172.055,51.424,160.365
C06812=1015.686,382.068,-157.567,172.065,51.422,160.367
C06813=1015.694,382.313,-157.608,172.076,51.420,160.368
C06814=1015.704,382.560,-157.648,172.085,51.418,160.369
C06815=1015.714,382.878,-157.702,172.099,51.415,160.371
C06816=1015.725,383.194,-157.755,172.112,51.412,160.373
C06817=1015.737,383.511,-157.807,172.125,51.410,160.374
C06818=1015.749,383.828,-157.860,172.139,51.407,160.376
C06819=1015.757,384.075,-157.901,172.149,51.405,160.378
C06820=1015.767,384.321,-157.943,172.159,51.403,160.379
C06821=1015.776,384.568,-157.984,172.170,51.401,160.380
C06822=1015.784,384.814,-158.025,172.180,51.399,160.382
C06823=1015.793,385.060,-158.067,172.191,51.396,160.383
C06824=1015.802,385.306,-158.108,172.201,51.395,160.385
C06825=1015.811,385.553,-158.150,172.212,51.393,160.386
C06826=1015.820,385.799,-158.192,172.222,51.391,160.387
C06827=1015.829,386.045,-158.233,172.233,51.389,160.389
C06828=1015.837,386.292,-158.275,172.244,51.387,160.391
C06829=1015.846,386.538,-158.317,172.255,51.385,160.392
C06830=1015.855,386.784,-158.359,172.264,51.383,160.393
C06831=1015.864,387.031,-158.400,172.276,51.381,160.395
C06832=1015.873,387.277,-158.442,172.287,51.379,160.396
C06833=1015.882,387.524,-158.484,172.297,51.378,160.398
C06834=1015.891,387.770,-158.525,172.308,51.376,160.399
C06835=1015.900,388.016,-158.568,172.319,51.374,160.401
C06836=1015.909,388.262,-158.610,172.330,51.373,160.403
C06837=1015.918,388.508,-158.651,172.340,51.371,160.404
C06838=1015.927,388.754,-158.694,172.351,51.369,160.406
C06839=1015.936,389.001,-158.735,172.362,51.367,160.407
C06840=1015.946,389.246,-158.778,172.373,51.366,160.409
C06841=1015.954,389.493,-158.820,172.384,51.364,160.410
C06842=1015.964,389.739,-158.863,172.395,51.362,160.412
C06843=1015.973,389.986,-158.905,172.405,51.360,160.413
C06844=1015.982,390.231,-158.947,172.417,51.359,160.415
C06845=1015.991,390.478,-158.989,172.428,51.357,160.416
C06846=1016.001,390.724,-159.032,172.439,51.355,160.418
C06847=1016.010,390.970,-159.074,172.449,51.353,160.419
C06848=1016.019,391.216,-159.116,172.461,51.352,160.421
C06849=1016.027,391.462,-159.159,172.472,51.350,160.423
C06850=1016.037,391.709,-159.202,172.483,51.348,160.424
C06851=1016.046,391.955,-159.244,172.494,51.347,160.426
C06852=1016.056,392.201,-159.287,172.505,51.345,160.428
C06853=1016.065,392.447,-159.330,172.517,51.344,160.429
C06854=1016.074,392.693,-159.372,172.528,51.342,160.431
C06855=1016.084,392.939,-159.415,172.538,51.341,160.433
C06856=1016.093,393.185,-159.458,172.550,51.340,160.434
C06857=1016.102,393.432,-159.501,172.561,51.338,160.436
C06858=1016.111,393.678,-159.543,172.573,51.336,160.438
C06859=1016.121,393.924,-159.586,172.585,51.335,160.440
C06860=1016.130,394.169,-159.630,172.596,51.333,160.441
C06861=1016.140,394.416,-159.673,172.607,51.332,160.443
C06862=1016.149,394.662,-159.715,172.619,51.331,160.445
C06863=1016.158,394.908,-159.759,172.630,51.330,160.446
C06864=1016.168,395.154,-159.802,172.641,51.328,160.448
C06865=1016.178,395.400,-159.845,172.652,51.326,160.450
C06866=1016.188,395.646,-159.888,172.664,51.325,160.451
C06867=1016.196,395.892,-159.931,172.675,51.324,160.453
C06868=1016.206,396.138,-159.975,172.687,51.322,160.455
C06869=1016.216,396.384,-160.017,172.699,51.321,160.457
C06870=1016.226,396.630,-160.061,172.710,51.319,160.459
C06871=1016.235,396.876,-160.104,172.722,51.318,160.460
C06872=1016.244,397.122,-160.148,172.733,51.317,160.462
C06873=1016.254,397.368,-160.192,172.746,51.316,160.464
C06874=1016.265,397.614,-160.235,172.757,51.315,160.466
C06875=1016.275,397.892,-160.284,172.771,51.313,160.468
C06876=1016.286,398.169,-160.334,172.784,51.311,160.470
C06877=1016.297,398.446,-160.383,172.798,51.310,160.472
C06878=1016.308,398.724,-160.432,172.811,51.309,160.474
C06879=1016.318,398.969,-160.476,172.823,51.308,160.476
C06880=1016.327,399.216,-160.520,172.834,51.307,160.478
C06881=1016.337,399.461,-160.563,172.846,51.305,160.480
C06882=1016.346,399.707,-160.607,172.859,51.304,160.482
C06883=1016.356,399.953,-160.651,172.870,51.303,160.483
C06884=1016.366,400.198,-160.696,172.882,51.302,160.485
C06885=1016.375,400.444,-160.740,172.895,51.301,160.487
C06886=1016.386,400.691,-160.784,172.906,51.300,160.489
C06887=1016.396,400.936,-160.828,172.919,51.299,160.491
C06888=1016.405,401.182,-160.873,172.931,51.298,160.493
C06889=1016.415,401.428,-160.917,172.943,51.297,160.495
C06890=1016.425,401.674,-160.961,172.955,51.296,160.497
C06891=1016.435,401.919,-161.006,172.968,51.295,160.499
C06892=1016.444,402.165,-161.050,172.980,51.294,160.501
C06893=1016.455,402.411,-161.094,172.992,51.293,160.503
C06894=1016.464,402.656,-161.139,173.005,51.292,160.505
C06895=1016.108,400.645,-161.119,172.888,51.366,160.504
C06896=1016.098,400.399,-161.075,172.876,51.367,160.502
C06897=1016.088,400.153,-161.032,172.863,51.368,160.500
C06898=1016.079,399.908,-160.987,172.852,51.370,160.498
C06899=1016.068,399.662,-160.943,172.840,51.370,160.496
C06900=1016.059,399.416,-160.899,172.828,51.372,160.495
C06901=1016.049,399.171,-160.855,172.816,51.374,160.493
C06902=1016.040,398.926,-160.812,172.804,51.374,160.491
C06903=1016.029,398.680,-160.769,172.792,51.376,160.489
C06904=1016.020,398.436,-160.724,172.780,51.377,160.487
C06905=1016.011,398.191,-160.681,172.768,51.378,160.485
C06906=1016.001,397.945,-160.638,172.757,51.379,160.483
C06907=1015.992,397.700,-160.595,172.744,51.381,160.481
C06908=1015.982,397.454,-160.551,172.733,51.382,160.480
C06909=1015.972,397.208,-160.507,172.721,51.384,160.478
C06910=1015.962,396.963,-160.464,172.709,51.385,160.476
C06911=1015.953,396.716,-160.421,172.698,51.386,160.474
C06912=1015.943,396.471,-160.377,172.686,51.388,160.473
C06913=1015.934,396.224,-160.334,172.675,51.389,160.471
C06914=1015.924,395.978,-160.290,172.663,51.391,160.469
C06915=1015.915,395.732,-160.248,172.651,51.392,160.467
C06916=1015.905,395.487,-160.204,172.640,51.393,160.465
C06917=1015.896,395.240,-160.161,172.629,51.395,160.464
C06918=1015.886,394.994,-160.118,172.617,51.397,160.462
C06919=1015.876,394.748,-160.075,172.605,51.398,160.460
C06920=1015.868,394.502,-160.032,172.594,51.399,160.459
C06921=1015.858,394.256,-159.989,172.583,51.401,160.457
C06922=1015.848,394.011,-159.946,172.571,51.403,160.455
C06923=1015.839,393.764,-159.902,172.559,51.404,160.453
C06924=1015.830,393.518,-159.860,172.548,51.406,160.452
C06925=1015.820,393.272,-159.817,172.537,51.407,160.450
C06926=1015.811,393.026,-159.775,172.525,51.409,160.449
C06927=1015.802,392.779,-159.731,172.514,51.411,160.447
C06928=1015.793,392.533,-159.689,172.503,51.413,160.445
C06929=1015.783,392.288,-159.647,172.492,51.413,160.443
C06930=1015.774,392.041,-159.603,172.481,51.415,160.442
C06931=1015.765,391.795,-159.561,172.470,51.417,160.440
C06932=1015.756,391.549,-159.518,172.458,51.419,160.439
C06933=1015.746,391.302,-159.476,172.447,51.421,160.437
C06934=1015.737,391.057,-159.434,172.436,51.423,160.435
C06935=1015.728,390.811,-159.391,172.425,51.424,160.434
C06936=1015.720,390.564,-159.349,172.414,51.426,160.432
C06937=1015.710,390.318,-159.306,172.403,51.427,160.431
C06938=1015.700,390.072,-159.264,172.391,51.429,160.429
C06939=1015.691,389.826,-159.222,172.380,51.431,160.428
C06940=1015.682,389.580,-159.180,172.370,51.433,160.426
C06941=1015.673,389.334,-159.138,172.359,51.435,160.424
C06942=1015.663,389.087,-159.095,172.348,51.437,160.423
C06943=1015.655,388.841,-159.053,172.337,51.438,160.421
C06944=1015.646,388.594,-159.012,172.326,51.440,160.420
C06945=1015.637,388.348,-158.969,172.315,51.442,160.418
C06946=1015.628,388.102,-158.927,172.305,51.444,160.417
C06947=1015.619,387.856,-158.885,172.294,51.446,160.415
C06948=1015.610,387.609,-158.844,172.282,51.448,160.414
C06949=1015.601,387.363,-158.801,172.272,51.449,160.412
C06950=1015.592,387.117,-158.759,172.261,51.452,160.411
C06951=1015.583,386.871,-158.718,172.250,51.454,160.409
C06952=1015.574,386.624,-158.676,172.240,51.455,160.408
C06953=1015.565,386.378,-158.634,172.229,51.458,160.406
C06954=1015.556,386.132,-158.593,172.219,51.459,160.405
C06955=1015.547,385.885,-158.551,172.208,51.461,160.403
C06956=1015.539,385.639,-158.509,172.197,51.464,160.402
C06957=1015.530,385.393,-158.467,172.187,51.465,160.401
C06958=1015.522,385.146,-158.427,172.176,51.468,160.399
C06959=1015.513,384.900,-158.385,172.166,51.470,160.398
C06960=1015.504,384.654,-158.343,172.155,51.472,160.396
C06961=1015.494,384.407,-158.302,172.145,51.474,160.395
C06962=1015.485,384.160,-158.261,172.134,51.476,160.394
C06963=1015.476,383.914,-158.219,172.124,51.478,160.392
C06964=1015.465,383.595,-158.167,172.110,51.481,160.391
C06965=1015.454,383.275,-158.113,172.097,51.484,160.389
C06966=1015.443,382.957,-158.060,172.084,51.487,160.387
C06967=1015.431,382.637,-158.007,172.069,51.490,160.385
C06968=1015.422,382.390,-157.966,172.060,51.492,160.384
C06969=1015.414,382.144,-157.926,172.050,51.494,160.383
C06970=1015.405,381.898,-157.884,172.039,51.496,160.381
C06971=1015.396,381.651,-157.843,172.029,51.498,160.380
C06972=1015.387,381.405,-157.803,172.018,51.501,160.378
C06973=1015.379,381.158,-157.762,172.008,51.503,160.377
C06974=1015.370,380.912,-157.721,171.997,51.505,160.376
C06975=1015.361,380.666,-157.680,171.988,51.508,160.375
C06976=1015.353,380.419,-157.640,171.978,51.510,160.373
C06977=1015.344,380.172,-157.599,171.967,51.512,160.372
C06978=1015.336,379.926,-157.558,171.957,51.514,160.371
C06979=1015.327,379.679,-157.518,171.948,51.517,160.370
C06980=1015.319,379.433,-157.477,171.937,51.520,160.368
C06981=1015.310,379.186,-157.436,171.927,51.522,160.367
C06982=1015.302,378.940,-157.395,171.917,51.524,160.366
C06983=1015.293,378.694,-157.355,171.907,51.527,160.364
C06984=1015.285,378.447,-157.314,171.897,51.529,160.363
C06985=1015.277,378.201,-157.274,171.887,51.531,160.362
C06986=1015.268,377.953,-157.234,171.878,51.534,160.361
C06987=1015.260,377.707,-157.193,171.867,51.536,160.360
C06988=1015.252,377.461,-157.153,171.857,51.539,160.358
C06989=1015.244,377.215,-157.112,171.848,51.541,160.357
C06990=1015.235,376.967,-157.072,171.838,51.544,160.356
C06991=1015.227,376.721,-157.032,171.827,51.546,160.355
C06992=1015.219,376.475,-156.991,171.818,51.549,160.354
C06993=1015.210,376.228,-156.952,171.808,51.551,160.353
C06994=1015.201,375.981,-156.911,171.798,51.553,160.351
C06995=1015.193,375.735,-156.870,171.789,51.556,160.350
C06996=1015.186,375.488,-156.830,171.779,51.558,160.349
C06997=1015.177,375.242,-156.790,171.769,51.562,160.348
C06998=1015.169,374.995,-156.750,171.760,51.564,160.347
C06999=1015.160,374.748,-156.711,171.750,51.566,160.345
C07000=1015.152,374.501,-156.671,171.740,51.569,160.344
C07001=1015.144,374.255,-156.631,171.731,51.572,160.343
C07002=1015.135,374.008,-156.591,171.721,51.575,160.342
C07003=1015.127,373.762,-156.552,171.711,51.577,160.341
C07004=1015.119,373.515,-156.512,171.701,51.580,160.340
C07005=1015.111,373.268,-156.473,171.692,51.583,160.339
C07006=1015.103,373.021,-156.433,171.683,51.586,160.338
C07007=1015.094,372.775,-156.393,171.673,51.588,160.337
C07008=1015.086,372.528,-156.354,171.664,51.591,160.336
C07009=1015.078,372.281,-156.314,171.654,51.594,160.335
C07010=1015.070,372.035,-156.275,171.645,51.597,160.334
C07011=1015.062,371.788,-156.235,171.635,51.600,160.332
C07012=1015.054,371.541,-156.196,171.625,51.603,160.331
C07013=1015.045,371.294,-156.156,171.616,51.605,160.330
C07014=1015.037,371.048,-156.116,171.606,51.608,160.329
C07015=1015.029,370.801,-156.077,171.597,51.611,160.328
C07016=1015.021,370.554,-156.038,171.588,51.614,160.327
C07017=1015.013,370.307,-155.999,171.578,51.616,160.326
C07018=1015.005,370.061,-155.960,171.569,51.619,160.325
C07019=1014.998,369.814,-155.920,171.559,51.622,160.324
C07020=1014.989,369.567,-155.881,171.551,51.625,160.323
C07021=1014.981,369.320,-155.842,171.541,51.628,160.322
C07022=1014.973,369.073,-155.802,171.532,51.631,160.321
C07023=1014.966,368.827,-155.764,171.522,51.634,160.320
C07024=1014.956,368.530,-155.716,171.511,51.637,160.319
C07025=1014.947,368.234,-155.670,171.501,51.641,160.318
C07026=1014.937,367.937,-155.622,171.490,51.644,160.317
C07027=1014.928,367.640,-155.575,171.478,51.648,160.315
C07028=1014.920,367.393,-155.536,171.469,51.651,160.314
C07029=1014.912,367.147,-155.497,171.460,51.654,160.314
C07030=1014.904,366.900,-155.459,171.450,51.657,160.312
C07031=1014.896,366.653,-155.420,171.441,51.660,160.312
C07032=1014.889,366.406,-155.381,171.433,51.663,160.311
C07033=1014.881,366.160,-155.342,171.424,51.666,160.310
C07034=1014.873,365.913,-155.304,171.415,51.669,160.309
C07035=1014.865,365.666,-155.265,171.406,51.672,160.308
C07036=1014.857,365.419,-155.227,171.397,51.676,160.307
C07037=1014.849,365.172,-155.188,171.388,51.679,160.306
C07038=1014.841,364.925,-155.150,171.378,51.682,160.305
C07039=1014.833,364.678,-155.112,171.369,51.685,160.304
C07040=1014.825,364.431,-155.073,171.360,51.688,160.304
C07041=1014.818,364.185,-155.035,171.351,51.692,160.303
C07042=1014.810,363.937,-154.996,171.343,51.694,160.302
C07043=1014.802,363.691,-154.958,171.334,51.698,160.301
C07044=1014.794,363.443,-154.920,171.325,51.701,160.300
C07045=1014.787,363.197,-154.882,171.316,51.704,160.299
C07046=1014.779,362.950,-154.843,171.307,51.708,160.298
C07047=1014.771,362.703,-154.805,171.298,51.711,160.298
C07048=1014.763,362.456,-154.767,171.289,51.714,160.296
C07049=1014.756,362.208,-154.729,171.281,51.717,160.296
C07050=1014.748,361.962,-154.690,171.272,51.720,160.295
C07051=1014.740,361.715,-154.652,171.263,51.724,160.294
C07052=1014.733,361.468,-154.614,171.254,51.727,160.293
C07053=1014.726,361.221,-154.575,171.245,51.731,160.292
C07054=1014.718,360.974,-154.537,171.237,51.734,160.292
C07055=1014.711,360.727,-154.500,171.228,51.737,160.291
C07056=1014.703,360.480,-154.461,171.219,51.741,160.290
C07057=1014.696,360.233,-154.424,171.210,51.744,160.289
C07058=1014.688,359.986,-154.385,171.202,51.747,160.289
C07059=1014.681,359.739,-154.348,171.193,51.751,160.288
C07060=1014.673,359.492,-154.309,171.184,51.754,160.287
C07061=1014.665,359.245,-154.272,171.175,51.758,160.286
C07062=1014.658,358.998,-154.234,171.168,51.761,160.286
C07063=1014.651,358.751,-154.196,171.159,51.765,160.285
C07064=1014.643,358.504,-154.158,171.150,51.768,160.284
C07065=1014.636,358.257,-154.121,171.141,51.771,160.283
C07066=1014.628,358.010,-154.084,171.133,51.775,160.282
C07067=1014.620,357.762,-154.046,171.124,51.778,160.282
C07068=1014.613,357.516,-154.008,171.116,51.783,160.281
C07069=1014.606,357.269,-153.970,171.108,51.786,160.280
C07070=1014.598,357.022,-153.933,171.099,51.789,160.279
C07071=1014.590,356.775,-153.896,171.090,51.793,160.279
C07072=1014.583,356.527,-153.858,171.081,51.796,160.278
C07073=1014.576,356.280,-153.821,171.074,51.800,160.277
C07074=1014.568,356.033,-153.784,171.065,51.803,160.276
C07075=1014.561,355.786,-153.746,171.056,51.807,160.276
C07076=1014.554,355.539,-153.709,171.049,51.811,160.275
C07077=1014.546,355.291,-153.672,171.040,51.814,160.274
C07078=1014.538,355.045,-153.635,171.031,51.819,160.274
C07079=1014.531,354.797,-153.597,171.023,51.822,160.273
C07080=1014.524,354.550,-153.560,171.014,51.826,160.272
C07081=1014.517,354.303,-153.522,171.006,51.830,160.272
C07082=1014.509,354.056,-153.486,170.998,51.833,160.271
C07083=1014.502,353.809,-153.449,170.989,51.837,160.270
C07084=1014.494,353.520,-153.406,170.980,51.841,160.270
C07085=1014.484,353.231,-153.362,170.970,51.845,160.269
C07086=1014.477,352.943,-153.319,170.961,51.850,160.268
C07087=1014.468,352.653,-153.276,170.951,51.854,160.268
C07088=1014.460,352.406,-153.239,170.943,51.858,160.267
C07089=1014.453,352.158,-153.202,170.934,51.862,160.266
C07090=1014.446,351.912,-153.166,170.926,51.866,160.266
C07091=1014.439,351.665,-153.129,170.917,51.869,160.265
C07092=1014.431,351.417,-153.092,170.909,51.873,160.264
C07093=1014.424,351.170,-153.055,170.901,51.877,160.264
C07094=1014.417,350.923,-153.019,170.893,51.881,160.263
C07095=1014.410,350.676,-152.982,170.885,51.885,160.263
C07096=1014.402,350.429,-152.945,170.877,51.889,160.262
C07097=1014.396,350.182,-152.909,170.868,51.893,160.261
C07098=1014.388,349.934,-152.873,170.861,51.897,160.261
C07099=1014.381,349.686,-152.836,170.852,51.901,160.260
C07100=1014.374,349.440,-152.799,170.845,51.905,160.260
C07101=1014.367,349.193,-152.762,170.836,51.909,160.259
C07102=1014.359,348.945,-152.726,170.828,51.913,160.258
C07103=1014.353,348.698,-152.690,170.820,51.917,160.258
C07104=1014.345,348.451,-152.653,170.812,51.921,160.257
C07105=1014.339,348.204,-152.617,170.804,51.925,160.257
C07106=1014.331,347.956,-152.581,170.796,51.929,160.256
C07107=1014.324,347.708,-152.544,170.788,51.933,160.256
C07108=1014.317,347.462,-152.508,170.780,51.937,160.255
C07109=1014.310,347.214,-152.471,170.773,51.941,160.255
C07110=1014.303,346.967,-152.435,170.764,51.945,160.254
C07111=1014.296,346.719,-152.399,170.756,51.949,160.254
C07112=1014.289,346.473,-152.363,170.748,51.953,160.253
C07113=1014.282,346.225,-152.326,170.741,51.957,160.253
C07114=1014.275,345.978,-152.290,170.732,51.961,160.252
C07115=1014.268,345.731,-152.255,170.724,51.966,160.252
C07116=1014.261,345.483,-152.219,170.716,51.970,160.251
C07117=1014.254,345.236,-152.182,170.708,51.974,160.251
C07118=1014.247,344.989,-152.146,170.701,51.978,160.250
C07119=1014.240,344.741,-152.111,170.693,51.983,160.250
C07120=1014.233,344.494,-152.074,170.685,51.986,160.249
C07121=1014.226,344.246,-152.039,170.677,51.991,160.249
C07122=1014.219,344.000,-152.003,170.670,51.995,160.248
C07123=1014.211,343.752,-151.967,170.661,51.999,160.248
C07124=1014.205,343.504,-151.931,170.654,52.004,160.247
C07125=1014.198,343.258,-151.895,170.645,52.008,160.247
C07126=1014.191,343.010,-151.860,170.638,52.012,160.246
C07127=1014.184,342.763,-151.824,170.630,52.017,160.246
C07128=1014.178,342.515,-151.788,170.623,52.021,160.246
C07129=1014.171,342.268,-151.752,170.614,52.025,160.245
C07130=1014.163,342.020,-151.717,170.607,52.029,160.245
C07131=1014.157,341.773,-151.682,170.599,52.034,160.244
C07132=1014.150,341.526,-151.646,170.592,52.038,160.244
